C03633=1021.085,424.714,339.079,174.416,50.425,160.512
C03634=1021.073,424.470,339.128,174.401,50.423,160.509
C03635=1021.061,424.224,339.178,174.386,50.421,160.506
C03636=1021.049,423.980,339.226,174.371,50.419,160.503
C03637=1021.037,423.735,339.276,174.356,50.417,160.500
C03638=1021.025,423.490,339.323,174.341,50.416,160.496
C03639=1021.013,423.245,339.372,174.326,50.414,160.493
C03640=1021.001,422.999,339.422,174.311,50.412,160.490
C03641=1020.989,422.755,339.470,174.297,50.410,160.487
C03642=1020.978,422.510,339.519,174.282,50.409,160.484
C03643=1020.966,422.265,339.567,174.267,50.407,160.481
C03644=1020.954,422.020,339.616,174.252,50.406,160.478
C03645=1020.942,421.775,339.664,174.237,50.404,160.475
C03646=1020.931,421.530,339.713,174.223,50.402,160.472
C03647=1020.920,421.285,339.761,174.209,50.400,160.469
C03648=1020.907,421.040,339.810,174.194,50.399,160.466
C03649=1020.895,420.794,339.858,174.179,50.397,160.463
C03650=1020.884,420.549,339.906,174.165,50.396,160.460
C03651=1020.872,420.304,339.954,174.150,50.395,160.458
C03652=1020.861,420.059,340.002,174.136,50.393,160.455
C03653=1020.849,419.814,340.050,174.122,50.391,160.452
C03654=1020.837,419.569,340.098,174.108,50.390,160.449
C03655=1020.826,419.324,340.146,174.094,50.388,160.446
C03656=1020.814,419.079,340.194,174.079,50.387,160.443
C03657=1020.803,418.833,340.241,174.065,50.386,160.440
C03658=1020.791,418.588,340.289,174.051,50.384,160.437
C03659=1020.780,418.343,340.337,174.037,50.383,160.435
C03660=1020.768,418.098,340.384,174.023,50.381,160.432
C03661=1020.757,417.853,340.433,174.009,50.380,160.429
C03662=1020.746,417.607,340.480,173.995,50.378,160.426
C03663=1020.734,417.362,340.527,173.981,50.377,160.423
C03664=1020.723,417.117,340.575,173.967,50.376,160.421
C03665=1020.712,416.872,340.622,173.954,50.374,160.418
C03666=1020.701,416.626,340.671,173.940,50.373,160.415
C03667=1020.690,416.381,340.717,173.926,50.372,160.412
C03668=1020.678,416.136,340.765,173.913,50.370,160.410
C03669=1020.667,415.890,340.813,173.898,50.369,160.407
C03670=1020.656,415.645,340.859,173.885,50.368,160.404
C03671=1020.644,415.400,340.907,173.872,50.366,160.401
C03672=1020.634,415.155,340.954,173.858,50.365,160.399
C03673=1020.623,414.909,341.001,173.844,50.364,160.396
C03674=1020.612,414.664,341.048,173.831,50.363,160.394
C03675=1020.600,414.419,341.095,173.818,50.362,160.391
C03676=1020.589,414.174,341.141,173.803,50.360,160.388
C03677=1020.578,413.928,341.188,173.790,50.359,160.386
C03678=1020.568,413.683,341.235,173.777,50.358,160.383
C03679=1020.556,413.437,341.282,173.764,50.357,160.381
C03680=1020.545,413.192,341.328,173.751,50.356,160.378
C03681=1020.535,412.947,341.375,173.738,50.355,160.375
C03682=1020.519,412.599,341.441,173.719,50.353,160.372
C03683=1020.503,412.251,341.507,173.700,50.352,160.368
C03684=1020.488,411.903,341.573,173.682,50.351,160.365
C03685=1020.472,411.556,341.639,173.663,50.349,160.361
C03686=1020.461,411.311,341.685,173.651,50.348,160.359
C03687=1020.451,411.065,341.731,173.637,50.347,160.356
C03688=1020.440,410.820,341.777,173.624,50.346,160.353
C03689=1020.430,410.574,341.824,173.611,50.345,160.351
C03690=1020.419,410.329,341.870,173.599,50.344,160.349
C03691=1020.409,410.083,341.916,173.586,50.343,160.346
C03692=1020.398,409.838,341.963,173.573,50.342,160.344
C03693=1020.387,409.592,342.009,173.561,50.341,160.341
C03694=1020.376,409.347,342.055,173.548,50.340,160.339
C03695=1020.366,409.101,342.100,173.535,50.340,160.336
C03696=1020.355,408.856,342.146,173.523,50.338,160.334
C03697=1020.345,408.610,342.192,173.510,50.338,160.332
C03698=1020.334,408.365,342.238,173.497,50.337,160.329
C03699=1020.323,408.119,342.284,173.484,50.336,160.327
C03700=1020.312,407.873,342.329,173.473,50.335,160.324
C03701=1020.302,407.627,342.375,173.460,50.335,160.322
C03702=1020.291,407.382,342.421,173.447,50.334,160.320
C03703=1020.281,407.137,342.466,173.434,50.334,160.317
C03704=1020.271,406.891,342.511,173.423,50.333,160.315
C03705=1020.259,406.645,342.557,173.410,50.332,160.313
C03706=1020.249,406.399,342.602,173.398,50.331,160.311
C03707=1020.239,406.154,342.647,173.386,50.331,160.308
C03708=1020.229,405.908,342.692,173.373,50.330,160.306
C03709=1020.217,405.663,342.738,173.361,50.329,160.304
C03710=1020.208,405.417,342.783,173.349,50.329,160.301
C03711=1020.197,405.172,342.829,173.337,50.328,160.299
C03712=1020.187,404.926,342.873,173.324,50.327,160.297
C03713=1020.177,404.680,342.919,173.313,50.327,160.295
C03714=1020.166,404.435,342.963,173.300,50.326,160.292
C03715=1020.156,404.189,343.009,173.288,50.325,160.290
C03716=1020.146,403.944,343.053,173.276,50.325,160.288
C03717=1020.136,403.697,343.099,173.264,50.324,160.286
C03718=1020.125,403.452,343.143,173.253,50.324,160.284
C03719=1020.115,403.206,343.188,173.240,50.323,160.281
C03720=1020.105,402.961,343.233,173.229,50.323,160.279
C03721=1020.096,402.715,343.278,173.216,50.323,160.277
C03722=1020.085,402.469,343.323,173.205,50.322,160.275
C03723=1020.075,402.224,343.367,173.193,50.321,160.273
C03724=1020.065,401.978,343.412,173.181,50.321,160.271
C03725=1020.055,401.733,343.457,173.169,50.320,160.268
C03726=1020.045,401.486,343.502,173.158,50.320,160.266
C03727=1020.035,401.241,343.546,173.147,50.320,160.264
C03728=1020.025,400.995,343.590,173.134,50.320,160.262
C03729=1020.016,400.750,343.635,173.123,50.319,160.260
C03730=1020.006,400.503,343.679,173.111,50.318,160.258
C03731=1019.995,400.257,343.724,173.100,50.318,160.256
C03732=1019.986,400.011,343.768,173.088,50.318,160.254
C03733=1019.976,399.766,343.813,173.076,50.318,160.252
C03734=1019.966,399.520,343.856,173.065,50.317,160.250
C03735=1019.956,399.275,343.901,173.054,50.317,160.248
C03736=1019.946,399.029,343.945,173.042,50.316,160.246
C03737=1019.937,398.783,343.989,173.031,50.316,160.244
C03738=1019.927,398.537,344.034,173.020,50.316,160.242
C03739=1019.917,398.291,344.077,173.008,50.316,160.240
C03740=1019.907,398.045,344.121,172.997,50.316,160.238
C03741=1019.897,397.799,344.165,172.985,50.316,160.236
C03742=1019.885,397.475,344.223,172.971,50.316,160.233
C03743=1019.872,397.150,344.280,172.955,50.315,160.231
C03744=1019.858,396.825,344.338,172.941,50.315,160.228
C03745=1019.846,396.500,344.396,172.926,50.315,160.226
C03746=1019.836,396.254,344.440,172.915,50.315,160.224
C03747=1019.826,396.009,344.483,172.904,50.315,160.222
C03748=1019.816,395.762,344.527,172.892,50.315,160.220
C03749=1019.807,395.516,344.570,172.882,50.315,160.218
C03750=1019.798,395.271,344.614,172.871,50.314,160.216
C03751=1019.788,395.025,344.657,172.860,50.314,160.214
C03752=1019.777,394.779,344.701,172.849,50.315,160.212
C03753=1019.768,394.532,344.744,172.838,50.315,160.211
C03754=1019.759,394.287,344.787,172.827,50.314,160.208
C03755=1019.749,394.041,344.830,172.816,50.314,160.207
C03756=1019.740,393.794,344.874,172.805,50.315,160.205
C03757=1019.730,393.549,344.917,172.794,50.315,160.203
C03758=1019.721,393.303,344.961,172.783,50.315,160.201
C03759=1019.711,393.056,345.003,172.773,50.315,160.200
C03760=1019.702,392.810,345.046,172.763,50.315,160.198
C03761=1019.692,392.564,345.090,172.751,50.315,160.196
C03762=1019.683,392.318,345.132,172.740,50.315,160.194
C03763=1019.673,392.072,345.175,172.730,50.316,160.192
C03764=1019.664,391.826,345.218,172.720,50.315,160.191
C03765=1019.655,391.580,345.261,172.709,50.316,160.189
C03766=1019.645,391.334,345.304,172.698,50.316,160.187
C03767=1019.636,391.088,345.347,172.687,50.316,160.185
C03768=1019.626,390.842,345.389,172.677,50.316,160.183
C03769=1019.616,390.596,345.432,172.667,50.317,160.182
C03770=1019.608,390.350,345.475,172.656,50.317,160.180
C03771=1019.599,390.103,345.517,172.645,50.317,160.178
C03772=1019.589,389.857,345.560,172.635,50.317,160.177
C03773=1019.580,389.611,345.602,172.624,50.318,160.175
C03774=1019.571,389.365,345.645,172.614,50.317,160.173
C03775=1019.562,389.119,345.688,172.604,50.318,160.171
C03776=1019.552,388.873,345.730,172.593,50.318,160.170
C03777=1019.543,388.627,345.772,172.583,50.319,160.168
C03778=1019.534,388.380,345.815,172.572,50.319,160.166
C03779=1019.524,388.134,345.857,172.562,50.320,160.165
C03780=1019.515,387.888,345.899,172.552,50.319,160.163
C03781=1019.506,387.642,345.942,172.541,50.320,160.161
C03782=1019.497,387.395,345.984,172.532,50.321,160.160
C03783=1019.488,387.149,346.027,172.521,50.321,160.158
C03784=1019.479,386.903,346.068,172.511,50.321,160.156
C03785=1019.470,386.656,346.110,172.501,50.322,160.155
C03786=1019.461,386.411,346.153,172.490,50.323,160.153
C03787=1019.452,386.164,346.194,172.481,50.323,160.152
C03788=1019.443,385.918,346.236,172.470,50.323,160.150
C03789=1019.434,385.672,346.278,172.460,50.324,160.148
C03790=1019.425,385.426,346.320,172.451,50.324,160.147
C03791=1019.416,385.179,346.362,172.440,50.325,160.145
C03792=1019.407,384.932,346.404,172.431,50.325,160.144
C03793=1019.397,384.686,346.445,172.420,50.326,160.142
C03794=1019.388,384.440,346.487,172.410,50.326,160.141
C03795=1019.379,384.194,346.528,172.400,50.327,160.139
C03796=1019.370,383.947,346.570,172.391,50.328,160.138
C03797=1019.361,383.701,346.612,172.380,50.329,160.136
C03798=1019.351,383.455,346.653,172.371,50.329,160.135
C03799=1019.343,383.209,346.694,172.360,50.330,160.133
C03800=1019.335,382.962,346.735,172.351,50.330,160.132
C03801=1019.326,382.716,346.777,172.341,50.331,160.130
C03802=1019.314,382.429,346.826,172.329,50.332,160.128
C03803=1019.304,382.141,346.873,172.318,50.333,160.127
C03804=1019.294,381.854,346.921,172.306,50.334,160.125
C03805=1019.283,381.567,346.970,172.296,50.335,160.123
C03806=1019.275,381.321,347.011,172.285,50.336,160.122
C03807=1019.266,381.074,347.052,172.276,50.336,160.120
C03808=1019.257,380.828,347.094,172.267,50.337,160.119
C03809=1019.248,380.581,347.135,172.256,50.338,160.117
C03810=1019.239,380.335,347.176,172.247,50.339,160.116
C03811=1019.231,380.088,347.217,172.238,50.340,160.115
C03812=1019.222,379.841,347.258,172.228,50.340,160.113
C03813=1019.214,379.596,347.299,172.218,50.341,160.112
C03814=1019.205,379.349,347.340,172.208,50.342,160.110
C03815=1019.196,379.102,347.380,172.199,50.343,160.109
C03816=1019.188,378.857,347.422,172.190,50.344,160.108
C03817=1019.179,378.610,347.463,172.180,50.344,160.106
C03818=1019.171,378.363,347.503,172.170,50.345,160.105
C03819=1019.162,378.117,347.545,172.161,50.346,160.103
C03820=1019.153,377.871,347.585,172.152,50.347,160.102
C03821=1019.145,377.624,347.626,172.143,50.348,160.101
C03822=1019.137,377.378,347.667,172.133,50.349,160.099
C03823=1019.128,377.131,347.708,172.123,50.350,160.098
C03824=1019.119,376.885,347.748,172.114,50.351,160.097
C03825=1019.110,376.638,347.789,172.105,50.352,160.095
C03826=1019.102,376.391,347.830,172.096,50.353,160.094
C03827=1019.094,376.144,347.871,172.087,50.354,160.093
C03828=1019.086,375.898,347.911,172.077,50.355,160.091
C03829=1019.076,375.651,347.952,172.068,50.356,160.090
C03830=1019.068,375.405,347.992,172.059,50.357,160.089
C03831=1019.060,375.159,348.032,172.050,50.358,160.087
C03832=1019.051,374.912,348.072,172.040,50.359,160.086
C03833=1019.043,374.666,348.113,172.031,50.361,160.085
C03834=1019.034,374.418,348.152,172.022,50.362,160.084
C03835=1019.025,374.172,348.193,172.013,50.363,160.082
C03836=1019.017,373.925,348.232,172.003,50.364,160.081
C03837=1019.009,373.679,348.273,171.995,50.365,160.080
C03838=1019.000,373.432,348.313,171.986,50.366,160.079
C03839=1018.991,373.186,348.353,171.976,50.367,160.077
C03840=1018.983,372.939,348.392,171.968,50.369,160.076
C03841=1018.974,372.692,348.433,171.958,50.370,160.075
C03842=1018.966,372.445,348.473,171.950,50.372,160.074
C03843=1018.958,372.199,348.513,171.940,50.372,160.072
C03844=1018.950,371.953,348.553,171.932,50.374,160.071
C03845=1018.941,371.706,348.592,171.923,50.375,160.070
C03846=1018.933,371.460,348.633,171.914,50.377,160.069
C03847=1018.924,371.212,348.672,171.905,50.378,160.068
C03848=1018.916,370.966,348.712,171.896,50.379,160.067
C03849=1018.908,370.719,348.752,171.887,50.380,160.065
C03850=1018.899,370.473,348.792,171.878,50.382,160.064
C03851=1018.892,370.226,348.832,171.869,50.383,160.063
C03852=1018.883,369.979,348.871,171.860,50.384,160.062
C03853=1018.876,369.732,348.911,171.851,50.386,160.061
C03854=1018.867,369.486,348.950,171.842,50.387,160.059
C03855=1018.859,369.239,348.990,171.834,50.388,160.058
C03856=1018.851,368.992,349.029,171.825,50.390,160.057
C03857=1018.842,368.746,349.069,171.817,50.391,160.056
C03858=1018.835,368.499,349.109,171.808,50.393,160.055
C03859=1018.826,368.252,349.148,171.799,50.394,160.054
C03860=1018.819,368.005,349.188,171.790,50.395,160.053
C03861=1018.810,367.759,349.227,171.781,50.397,160.051
C03862=1018.801,367.494,349.269,171.772,50.398,160.050
C03863=1018.793,367.229,349.311,171.763,50.400,160.049
C03864=1018.784,366.963,349.353,171.754,50.402,160.048
C03865=1018.775,366.699,349.396,171.745,50.404,160.047
C03866=1018.767,366.452,349.434,171.736,50.405,160.046
C03867=1018.759,366.205,349.473,171.727,50.407,160.045
C03868=1018.750,365.958,349.512,171.719,50.408,160.044
C03869=1018.743,365.712,349.551,171.710,50.410,160.043
C03870=1018.734,365.465,349.590,171.701,50.411,160.041
C03871=1018.727,365.218,349.630,171.693,50.413,160.040
C03872=1018.719,364.971,349.668,171.685,50.415,160.040
C03873=1018.710,364.724,349.707,171.676,50.416,160.038
C03874=1018.703,364.477,349.746,171.667,50.418,160.037
C03875=1018.694,364.230,349.784,171.659,50.420,160.036
C03876=1018.686,363.984,349.824,171.651,50.421,160.035
C03877=1018.678,363.737,349.862,171.642,50.423,160.034
C03878=1018.670,363.490,349.900,171.634,50.425,160.033
C03879=1018.662,363.243,349.940,171.625,50.427,160.032
C03880=1018.654,362.997,349.978,171.617,50.428,160.031
C03881=1018.647,362.749,350.017,171.609,50.430,160.030
C03882=1018.639,362.502,350.056,171.600,50.432,160.029
C03883=1018.631,362.256,350.094,171.591,50.433,160.028
C03884=1018.623,362.009,350.133,171.584,50.435,160.027
C03885=1018.615,361.762,350.172,171.575,50.437,160.026
C03886=1018.607,361.515,350.210,171.567,50.439,160.025
C03887=1018.599,361.268,350.249,171.560,50.441,160.025
C03888=1018.591,361.022,350.287,171.551,50.442,160.023
C03889=1018.583,360.774,350.326,171.542,50.445,160.023
C03890=1018.577,360.563,350.359,171.536,50.445,160.022
C03891=1018.571,360.352,350.391,171.528,50.447,160.021
C03892=1018.564,360.142,350.425,171.522,50.449,160.020
C03893=1018.557,359.931,350.457,171.514,50.451,160.019
C03894=1018.550,359.720,350.490,171.508,50.452,160.019
C03895=1018.544,359.509,350.522,171.501,50.454,160.018
C03896=1018.538,359.299,350.555,171.494,50.455,160.017
C03897=1018.531,359.088,350.587,171.487,50.457,160.016
C03898=1018.523,358.841,350.625,171.478,50.459,160.015
C03899=1018.515,358.595,350.664,171.471,50.461,160.014
C03900=1018.507,358.347,350.702,171.462,50.463,160.013
C03901=1018.500,358.100,350.740,171.455,50.465,160.013
C03902=1018.492,357.853,350.778,171.446,50.467,160.012
C03903=1018.484,357.606,350.816,171.438,50.469,160.011
C03904=1018.476,357.360,350.854,171.431,50.471,160.010
C03905=1018.468,357.112,350.892,171.422,50.473,160.009
C03906=1018.461,356.865,350.930,171.414,50.475,160.008
C03907=1018.453,356.618,350.967,171.406,50.477,160.007
C03908=1018.445,356.371,351.006,171.398,50.479,160.006
C03909=1018.437,356.124,351.043,171.391,50.481,160.006
C03910=1018.430,355.877,351.080,171.382,50.483,160.005
C03911=1018.423,355.631,351.119,171.374,50.485,160.004
C03912=1018.415,355.383,351.157,171.366,50.487,160.003
C03913=1018.407,355.136,351.193,171.358,50.490,160.002
C03914=1018.399,354.889,351.232,171.351,50.492,160.001
C03915=1018.392,354.642,351.269,171.343,50.494,160.001
C03916=1018.385,354.395,351.307,171.335,50.496,160.000
C03917=1018.376,354.148,351.344,171.327,50.498,159.999
C03918=1018.369,353.900,351.382,171.320,50.501,159.998
C03919=1018.361,353.654,351.420,171.311,50.503,159.997
C03920=1018.354,353.407,351.457,171.304,50.505,159.997
C03921=1018.346,353.160,351.494,171.296,50.508,159.996
C03922=1018.336,352.830,351.543,171.286,50.510,159.995
C03923=1018.326,352.500,351.594,171.275,50.513,159.994
C03924=1018.315,352.170,351.644,171.265,50.516,159.993
C03925=1018.305,351.840,351.694,171.255,50.520,159.992
C03926=1018.298,351.592,351.730,171.246,50.522,159.991
C03927=1018.290,351.346,351.767,171.239,50.524,159.990
C03928=1018.283,351.098,351.805,171.231,50.527,159.989
C03929=1018.276,350.851,351.842,171.224,50.529,159.989
C03930=1018.268,350.604,351.879,171.216,50.531,159.988
C03931=1018.261,350.357,351.916,171.209,50.534,159.987
C03932=1018.253,350.110,351.953,171.200,50.536,159.986
C03933=1018.246,349.863,351.991,171.193,50.538,159.986
C03934=1018.238,349.616,352.027,171.185,50.541,159.985
C03935=1018.231,349.368,352.064,171.178,50.543,159.984
C03936=1018.223,349.121,352.102,171.171,50.545,159.984
C03937=1018.216,348.874,352.138,171.163,50.548,159.983
C03938=1018.209,348.627,352.175,171.156,50.551,159.982
C03939=1018.201,348.380,352.212,171.147,50.553,159.981
C03940=1018.194,348.133,352.249,171.140,50.555,159.981
C03941=1018.186,347.886,352.286,171.132,50.558,159.980
C03942=1018.179,347.638,352.323,171.125,50.561,159.980
C03943=1018.171,347.391,352.360,171.118,50.563,159.979
C03944=1018.165,347.144,352.396,171.110,50.565,159.978
C03945=1018.157,346.897,352.433,171.103,50.568,159.977
C03946=1018.150,346.650,352.470,171.095,50.571,159.977
C03947=1018.142,346.402,352.506,171.088,50.573,159.976
C03948=1018.135,346.155,352.542,171.080,50.576,159.975
C03949=1018.128,345.908,352.579,171.073,50.578,159.975
C03950=1018.120,345.661,352.616,171.066,50.581,159.974
C03951=1018.113,345.413,352.652,171.058,50.584,159.973
C03952=1018.106,345.166,352.688,171.051,50.586,159.973
C03953=1018.099,344.919,352.725,171.043,50.589,159.972
C03954=1018.091,344.672,352.761,171.036,50.592,159.972
C03955=1018.083,344.425,352.798,171.029,50.594,159.971
C03956=1018.077,344.178,352.834,171.021,50.597,159.970
C03957=1018.069,343.930,352.870,171.014,50.600,159.970
C03958=1018.061,343.683,352.907,171.006,50.603,159.969
C03959=1018.055,343.436,352.943,170.999,50.605,159.969
C03960=1018.047,343.188,352.979,170.992,50.608,159.968
C03961=1018.040,342.941,353.015,170.984,50.611,159.967
C03962=1018.033,342.694,353.052,170.977,50.613,159.967
C03963=1018.026,342.446,353.088,170.970,50.616,159.966
C03964=1018.018,342.199,353.124,170.963,50.619,159.966
C03965=1018.011,341.951,353.159,170.956,50.622,159.965
C03966=1018.005,341.704,353.196,170.949,50.624,159.964
C03967=1017.997,341.457,353.232,170.941,50.628,159.964
C03968=1017.990,341.210,353.268,170.934,50.630,159.963
C03969=1017.982,340.963,353.304,170.927,50.633,159.963
C03970=1017.976,340.715,353.339,170.920,50.636,159.962
C03971=1017.969,340.468,353.376,170.913,50.639,159.962
C03972=1017.962,340.221,353.412,170.906,50.642,159.961
C03973=1017.954,339.973,353.448,170.898,50.645,159.961
C03974=1017.947,339.726,353.483,170.891,50.648,159.960
C03975=1017.939,339.479,353.520,170.884,50.650,159.960
C03976=1017.933,339.231,353.555,170.877,50.654,159.959
C03977=1017.926,338.984,353.591,170.870,50.656,159.958
C03978=1017.919,338.737,353.627,170.863,50.659,159.958
C03979=1017.912,338.489,353.662,170.855,50.663,159.958
C03980=1017.905,338.241,353.698,170.848,50.665,159.957
C03981=1017.897,337.995,353.734,170.842,50.668,159.956
C03982=1017.890,337.735,353.771,170.834,50.672,159.956
C03983=1017.883,337.474,353.808,170.826,50.674,159.955
C03984=1017.875,337.214,353.845,170.819,50.678,159.955
C03985=1017.867,336.953,353.883,170.812,50.681,159.954
C03986=1017.860,336.706,353.918,170.805,50.684,159.954
C03987=1017.853,336.459,353.953,170.798,50.688,159.953
C03988=1017.846,336.211,353.989,170.791,50.690,159.953
C03989=1017.839,335.964,354.025,170.784,50.693,159.952
C03990=1017.832,335.717,354.060,170.776,50.697,159.952
C03991=1017.825,335.469,354.095,170.770,50.700,159.952
C03992=1017.818,335.221,354.131,170.763,50.703,159.951
C03993=1017.811,334.974,354.166,170.756,50.706,159.951
C03994=1017.804,334.727,354.202,170.749,50.709,159.950
C03995=1017.797,334.480,354.237,170.742,50.713,159.950
C03996=1017.790,334.232,354.272,170.736,50.716,159.949
C03997=1017.783,333.984,354.307,170.729,50.719,159.949
C03998=1017.777,333.737,354.342,170.721,50.722,159.949
C03999=1017.770,333.490,354.378,170.715,50.725,159.948
C04000=1017.763,333.242,354.413,170.708,50.728,159.948
C04001=1017.756,332.995,354.448,170.702,50.732,159.947
C04002=1017.749,332.747,354.483,170.694,50.735,159.947
C04003=1017.741,332.500,354.518,170.687,50.738,159.946
C04004=1017.735,332.252,354.553,170.681,50.741,159.946
C04005=1017.728,332.005,354.588,170.674,50.744,159.946
C04006=1017.721,331.757,354.623,170.666,50.748,159.945
C04007=1017.714,331.510,354.657,170.660,50.752,159.945
C04008=1017.707,331.263,354.692,170.654,50.755,159.944
C04009=1017.700,331.015,354.727,170.647,50.758,159.944
C04010=1017.693,330.768,354.761,170.639,50.761,159.944
C04011=1017.686,330.520,354.796,170.633,50.765,159.943
C04012=1017.680,330.273,354.831,170.626,50.768,159.943
C04013=1017.672,330.025,354.865,170.620,50.771,159.943
C04014=1017.666,329.778,354.900,170.613,50.775,159.942
C04015=1017.659,329.530,354.936,170.606,50.779,159.942
C04016=1017.652,329.282,354.970,170.599,50.782,159.941
C04017=1017.645,329.035,355.005,170.593,50.785,159.941
C04018=1017.638,328.787,355.039,170.586,50.789,159.941
C04019=1017.632,328.540,355.074,170.579,50.792,159.940
C04020=1017.624,328.292,355.108,170.573,50.796,159.940
C04021=1017.618,328.045,355.143,170.566,50.799,159.940
C04022=1017.611,327.797,355.177,170.560,50.803,159.939
C04023=1017.604,327.550,355.212,170.552,50.806,159.939
C04024=1017.598,327.303,355.246,170.546,50.810,159.939
C04025=1017.591,327.055,355.281,170.539,50.813,159.938
C04026=1017.584,326.808,355.315,170.533,50.817,159.938
C04027=1017.577,326.560,355.349,170.526,50.820,159.938
C04028=1017.571,326.312,355.385,170.519,50.824,159.937
C04029=1017.563,326.065,355.418,170.513,50.828,159.937
C04030=1017.557,325.818,355.452,170.506,50.831,159.937
C04031=1017.550,325.570,355.486,170.500,50.835,159.937
C04032=1017.543,325.322,355.520,170.493,50.839,159.936
C04033=1017.536,325.075,355.555,170.487,50.843,159.936
C04034=1017.529,324.827,355.588,170.480,50.846,159.936
C04035=1017.522,324.579,355.623,170.474,50.849,159.935
C04036=1017.515,324.332,355.656,170.467,50.854,159.935
C04037=1017.508,324.085,355.690,170.460,50.857,159.935
C04038=1017.501,323.837,355.724,170.454,50.861,159.935
C04039=1017.495,323.589,355.758,170.448,50.865,159.935
C04040=1017.488,323.342,355.792,170.441,50.869,159.934
C04041=1017.481,323.094,355.825,170.434,50.872,159.934
C04042=1017.474,322.829,355.862,170.427,50.877,159.934
C04043=1017.466,322.565,355.898,170.421,50.881,159.934
C04044=1017.459,322.300,355.934,170.414,50.885,159.933
C04045=1017.452,322.035,355.970,170.407,50.889,159.933
C04046=1017.445,321.788,356.004,170.400,50.893,159.933
C04047=1017.438,321.540,356.037,170.394,50.896,159.933
C04048=1017.431,321.292,356.071,170.388,50.900,159.932
C04049=1017.425,321.045,356.105,170.381,50.904,159.932
C04050=1017.418,320.798,356.139,170.375,50.908,159.932
C04051=1017.412,320.550,356.171,170.368,50.912,159.932
C04052=1017.405,320.302,356.205,170.362,50.916,159.931
C04053=1017.397,320.055,356.239,170.356,50.919,159.931
C04054=1017.392,319.807,356.273,170.349,50.924,159.931
C04055=1017.385,319.559,356.306,170.342,50.927,159.931
C04056=1017.378,319.312,356.340,170.337,50.932,159.931
C04057=1017.371,319.064,356.373,170.330,50.936,159.930
C04058=1017.365,318.816,356.407,170.324,50.939,159.930
C04059=1017.358,318.569,356.441,170.317,50.943,159.930
C04060=1017.352,318.321,356.473,170.311,50.947,159.930
C04061=1017.345,318.074,356.507,170.305,50.952,159.930
C04062=1017.339,317.826,356.541,170.299,50.955,159.930
C04063=1017.332,317.578,356.574,170.292,50.959,159.929
C04064=1017.325,317.331,356.608,170.286,50.963,159.929
C04065=1017.318,317.083,356.641,170.279,50.968,159.929
C04066=1017.312,316.836,356.674,170.273,50.972,159.929
C04067=1017.306,316.588,356.708,170.267,50.975,159.929
C04068=1017.299,316.340,356.741,170.261,50.980,159.929
C04069=1017.293,316.093,356.774,170.255,50.984,159.928
C04070=1017.286,315.844,356.807,170.249,50.987,159.928
C04071=1017.280,315.597,356.841,170.242,50.992,159.928
C04072=1017.274,315.349,356.874,170.236,50.996,159.928
C04073=1017.267,315.101,356.907,170.230,51.000,159.928
C04074=1017.260,314.854,356.941,170.224,51.004,159.928
C04075=1017.254,314.607,356.974,170.217,51.008,159.927
C04076=1017.248,314.359,357.007,170.212,51.012,159.927
C04077=1017.241,314.111,357.041,170.205,51.016,159.927
C04078=1017.235,313.863,357.073,170.198,51.021,159.927
C04079=1017.229,313.616,357.106,170.192,51.025,159.927
C04080=1017.221,313.368,357.140,170.186,51.029,159.927
C04081=1017.216,313.120,357.173,170.180,51.033,159.927
C04082=1017.209,312.873,357.206,170.174,51.037,159.927
C04083=1017.203,312.625,357.239,170.169,51.042,159.927
C04084=1017.197,312.377,357.272,170.162,51.046,159.926
C04085=1017.190,312.130,357.305,170.157,51.050,159.926
C04086=1017.184,311.882,357.339,170.150,51.054,159.926
C04087=1017.178,311.634,357.371,170.143,51.059,159.926
C04088=1017.172,311.387,357.404,170.138,51.063,159.926
C04089=1017.165,311.139,357.437,170.131,51.067,159.926
C04090=1017.159,310.891,357.470,170.126,51.071,159.926
C04091=1017.153,310.644,357.503,170.120,51.076,159.926
C04092=1017.147,310.395,357.536,170.114,51.080,159.926
C04093=1017.140,310.148,357.569,170.108,51.084,159.926
C04094=1017.134,309.900,357.602,170.102,51.089,159.926
C04095=1017.128,309.652,357.634,170.096,51.092,159.925
C04096=1017.121,309.405,357.667,170.089,51.097,159.925
C04097=1017.115,309.157,357.700,170.083,51.102,159.925
C04098=1017.108,308.909,357.731,170.077,51.106,159.925
C04099=1017.102,308.662,357.764,170.071,51.110,159.925
C04100=1017.095,308.415,357.796,170.066,51.115,159.925
C04101=1017.089,308.166,357.828,170.059,51.120,159.925
C04102=1017.082,307.907,357.862,170.053,51.125,159.925
C04103=1017.075,307.648,357.896,170.047,51.130,159.925
C04104=1017.068,307.389,357.929,170.041,51.134,159.925
C04105=1017.061,307.130,357.963,170.034,51.139,159.925
C04106=1017.055,306.882,357.995,170.028,51.143,159.925
C04107=1017.048,306.634,358.028,170.022,51.148,159.925
C04108=1017.042,306.386,358.060,170.017,51.153,159.925
C04109=1017.035,306.139,358.092,170.010,51.158,159.925
C04110=1017.029,305.891,358.124,170.004,51.162,159.925
C04111=1017.022,305.643,358.156,169.998,51.167,159.925
C04112=1017.016,305.395,358.188,169.993,51.171,159.925
C04113=1017.010,305.147,358.220,169.987,51.176,159.925
C04114=1017.003,304.900,358.252,169.980,51.181,159.925
C04115=1016.997,304.651,358.284,169.975,51.186,159.925
C04116=1016.990,304.404,358.316,169.969,51.190,159.925
C04117=1016.984,304.156,358.348,169.963,51.195,159.925
C04118=1016.977,303.908,358.380,169.958,51.200,159.925
C04119=1016.971,303.660,358.412,169.951,51.204,159.925
C04120=1016.965,303.412,358.445,169.945,51.209,159.925
C04121=1016.959,303.165,358.476,169.940,51.214,159.925
C04122=1016.953,302.917,358.508,169.934,51.218,159.925
C04123=1016.946,302.670,358.540,169.928,51.223,159.925
C04124=1016.940,302.421,358.572,169.921,51.228,159.926
C04125=1016.933,302.173,358.603,169.916,51.233,159.926
C04126=1016.927,301.925,358.635,169.910,51.238,159.926
C04127=1016.920,301.677,358.667,169.904,51.243,159.926
C04128=1016.915,301.430,358.698,169.899,51.247,159.926
C04129=1016.908,301.183,358.731,169.893,51.252,159.926
C04130=1016.902,300.934,358.763,169.886,51.257,159.926
C04131=1016.896,300.686,358.795,169.881,51.262,159.926
C04132=1016.889,300.438,358.826,169.875,51.267,159.926
C04133=1016.884,300.191,358.858,169.870,51.272,159.926
C04134=1016.877,299.943,358.889,169.864,51.276,159.926
C04135=1016.871,299.695,358.921,169.859,51.281,159.926
C04136=1016.865,299.447,358.953,169.852,51.286,159.926
C04137=1016.859,299.199,358.984,169.846,51.291,159.926
C04138=1016.852,298.951,359.016,169.841,51.296,159.927
C04139=1016.846,298.703,359.048,169.835,51.301,159.927
C04140=1016.840,298.455,359.079,169.830,51.306,159.927
C04141=1016.834,298.208,359.111,169.824,51.311,159.927
C04142=1016.828,297.959,359.143,169.818,51.316,159.927
C04143=1016.822,297.712,359.174,169.812,51.321,159.927
C04144=1016.816,297.464,359.206,169.806,51.326,159.927
C04145=1016.809,297.216,359.237,169.801,51.331,159.927
C04146=1016.803,296.968,359.269,169.796,51.336,159.927
C04147=1016.798,296.720,359.300,169.790,51.340,159.927
C04148=1016.792,296.472,359.332,169.783,51.346,159.927
C04149=1016.786,296.225,359.363,169.778,51.351,159.928
C04150=1016.780,295.976,359.395,169.772,51.356,159.928
C04151=1016.773,295.729,359.426,169.767,51.361,159.928
C04152=1016.767,295.481,359.458,169.761,51.366,159.928
C04153=1016.761,295.233,359.489,169.756,51.371,159.928
C04154=1016.756,294.985,359.520,169.751,51.376,159.928
C04155=1016.750,294.737,359.552,169.744,51.381,159.928
C04156=1016.744,294.490,359.583,169.738,51.386,159.928
C04157=1016.738,294.241,359.615,169.733,51.391,159.929
C04158=1016.732,293.997,359.646,169.728,51.396,159.929
C04159=1016.726,293.752,359.676,169.722,51.402,159.929
C04160=1016.720,293.507,359.707,169.716,51.406,159.929
C04161=1016.714,293.262,359.739,169.711,51.411,159.929
C04162=1016.708,293.018,359.769,169.706,51.416,159.929
C04163=1016.702,292.773,359.800,169.700,51.422,159.930
C04164=1016.696,292.529,359.830,169.695,51.427,159.930
C04165=1016.690,292.284,359.861,169.689,51.432,159.930
C04166=1016.684,292.037,359.892,169.683,51.437,159.930
C04167=1016.678,291.789,359.922,169.678,51.443,159.930
C04168=1016.672,291.540,359.954,169.672,51.448,159.930
C04169=1016.666,291.293,359.985,169.667,51.453,159.931
C04170=1016.660,291.044,360.016,169.662,51.459,159.931
C04171=1016.654,290.796,360.046,169.655,51.464,159.931
C04172=1016.647,290.548,360.077,169.650,51.469,159.931
C04173=1016.641,290.301,360.108,169.645,51.475,159.932
C04174=1016.636,290.053,360.138,169.639,51.480,159.932
C04175=1016.629,289.804,360.169,169.633,51.486,159.932
C04176=1016.623,289.557,360.200,169.628,51.491,159.932
C04177=1016.617,289.309,360.231,169.622,51.496,159.932
C04178=1016.612,289.060,360.262,169.617,51.501,159.933
C04179=1016.606,288.813,360.292,169.611,51.508,159.933
C04180=1016.599,288.564,360.323,169.606,51.513,159.933
C04181=1016.593,288.316,360.353,169.600,51.518,159.933
C04182=1016.587,288.068,360.384,169.595,51.524,159.934
C04183=1016.581,287.821,360.415,169.589,51.529,159.934
C04184=1016.575,287.573,360.445,169.584,51.534,159.934
C04185=1016.569,287.324,360.476,169.579,51.540,159.934
C04186=1016.563,287.076,360.506,169.573,51.545,159.934
C04187=1016.557,286.829,360.536,169.567,51.552,159.935
C04188=1016.551,286.580,360.567,169.562,51.557,159.935
C04189=1016.545,286.332,360.598,169.557,51.563,159.935
C04190=1016.539,286.084,360.628,169.552,51.568,159.936
C04191=1016.533,285.837,360.658,169.546,51.574,159.936
C04192=1016.527,285.588,360.689,169.540,51.579,159.936
C04193=1016.521,285.340,360.719,169.535,51.585,159.936
C04194=1016.515,285.092,360.749,169.530,51.590,159.937
C04195=1016.509,284.843,360.780,169.524,51.596,159.937
C04196=1016.503,284.595,360.810,169.518,51.602,159.937
C04197=1016.497,284.348,360.840,169.513,51.608,159.938
C04198=1016.491,284.100,360.870,169.508,51.613,159.938
C04199=1016.485,283.852,360.900,169.502,51.619,159.938
C04200=1016.479,283.603,360.930,169.497,51.625,159.938
C04201=1016.472,283.356,360.960,169.492,51.631,159.939
C04202=1016.467,283.107,360.990,169.486,51.636,159.939
C04203=1016.461,282.859,361.020,169.481,51.642,159.939
C04204=1016.455,282.611,361.051,169.476,51.648,159.940
C04205=1016.448,282.363,361.080,169.470,51.653,159.940
C04206=1016.443,282.115,361.110,169.465,51.659,159.940
C04207=1016.437,281.867,361.141,169.460,51.665,159.941
C04208=1016.431,281.619,361.170,169.455,51.671,159.941
C04209=1016.425,281.371,361.200,169.449,51.677,159.941
C04210=1016.419,281.122,361.230,169.443,51.682,159.941
C04211=1016.413,280.874,361.260,169.438,51.688,159.942
C04212=1016.406,280.626,361.289,169.432,51.695,159.942
C04213=1016.401,280.378,361.320,169.427,51.700,159.942
C04214=1016.395,280.130,361.349,169.422,51.706,159.943
C04215=1016.389,279.882,361.380,169.417,51.713,159.943
C04216=1016.383,279.634,361.409,169.412,51.718,159.944
C04217=1016.377,279.386,361.439,169.407,51.724,159.944
C04218=1016.371,279.168,361.465,169.401,51.729,159.944
C04219=1016.367,278.951,361.492,169.397,51.734,159.944
C04220=1016.362,278.734,361.518,169.393,51.740,159.945
C04221=1016.356,278.517,361.544,169.388,51.745,159.945
C04222=1016.351,278.300,361.569,169.383,51.750,159.945
C04223=1016.347,278.083,361.596,169.378,51.756,159.946
C04224=1016.341,277.866,361.622,169.374,51.761,159.946
C04225=1016.332,277.478,361.668,169.366,51.770,159.947
C04226=1016.326,277.230,361.698,169.360,51.776,159.947
C04227=1016.321,276.982,361.728,169.355,51.782,159.947
C04228=1016.315,276.733,361.757,169.350,51.788,159.948
C04229=1016.309,276.486,361.787,169.344,51.794,159.948
C04230=1016.303,276.237,361.817,169.339,51.800,159.948
C04231=1016.298,275.989,361.846,169.334,51.806,159.949
C04232=1016.291,275.741,361.875,169.328,51.812,159.949
C04233=1016.285,275.493,361.905,169.324,51.819,159.950
C04234=1016.279,275.245,361.935,169.319,51.825,159.950
C04235=1016.273,274.996,361.964,169.313,51.831,159.950
C04236=1016.268,274.748,361.993,169.308,51.837,159.951
C04237=1016.261,274.500,362.022,169.303,51.844,159.951
C04238=1016.256,274.251,362.052,169.298,51.850,159.952
C04239=1016.250,274.003,362.081,169.293,51.855,159.952
C04240=1016.244,273.755,362.111,169.287,51.862,159.953
C04241=1016.238,273.507,362.139,169.282,51.868,159.953
C04242=1016.233,273.259,362.169,169.277,51.874,159.953
C04243=1016.227,273.011,362.198,169.272,51.881,159.954
C04244=1016.221,272.762,362.228,169.267,51.887,159.954
C04245=1016.215,272.514,362.257,169.261,51.893,159.955
C04246=1016.209,272.266,362.286,169.256,51.900,159.955
C04247=1016.203,272.018,362.315,169.251,51.906,159.956
C04248=1016.197,271.770,362.345,169.246,51.912,159.956
C04249=1016.192,271.522,362.374,169.241,51.919,159.956
C04250=1016.186,271.274,362.403,169.235,51.925,159.957
C04251=1016.180,271.025,362.432,169.231,51.931,159.957
C04252=1016.174,270.777,362.461,169.226,51.937,159.958
C04253=1016.168,270.528,362.490,169.220,51.944,159.958
C04254=1016.162,270.280,362.519,169.215,51.950,159.959
C04255=1016.157,270.033,362.548,169.210,51.957,159.959
C04256=1016.151,269.784,362.577,169.205,51.963,159.960
C04257=1016.145,269.535,362.606,169.199,51.970,159.960
C04258=1016.139,269.287,362.635,169.195,51.977,159.961
C04259=1016.134,269.039,362.664,169.190,51.982,159.961
C04260=1016.128,268.791,362.693,169.184,51.989,159.962
C04261=1016.122,268.543,362.722,169.179,51.995,159.962
C04262=1016.116,268.294,362.751,169.174,52.002,159.962
C04263=1016.111,268.047,362.780,169.169,52.009,159.963
C04264=1016.105,267.798,362.808,169.164,52.016,159.964
C04265=1016.099,267.550,362.837,169.159,52.022,159.964
C04266=1016.093,267.301,362.866,169.153,52.029,159.964
C04267=1016.087,267.054,362.894,169.149,52.035,159.965
C04268=1016.082,266.805,362.923,169.144,52.041,159.965
C04269=1016.076,266.556,362.952,169.138,52.048,159.966
C04270=1016.070,266.308,362.980,169.134,52.055,159.967
C04271=1016.064,266.060,363.009,169.128,52.062,159.967
C04272=1016.058,265.812,363.038,169.124,52.068,159.968
C04273=1016.053,265.564,363.067,169.118,52.075,159.968
C04274=1016.047,265.315,363.095,169.114,52.081,159.969
C04275=1016.041,265.067,363.124,169.108,52.088,159.969
C04276=1016.036,264.819,363.152,169.104,52.095,159.970
C04277=1016.029,264.571,363.181,169.098,52.102,159.970
C04278=1016.025,264.334,363.208,169.094,52.108,159.971
C04279=1016.018,264.098,363.235,169.089,52.114,159.971
C04280=1016.013,263.862,363.262,169.084,52.121,159.972
C04281=1016.008,263.625,363.290,169.080,52.127,159.972
C04282=1016.002,263.389,363.317,169.074,52.134,159.973
C04283=1015.997,263.153,363.344,169.069,52.140,159.973
C04284=1015.991,262.916,363.371,169.065,52.147,159.974
C04285=1015.986,262.680,363.398,169.060,52.154,159.974
C04286=1015.980,262.432,363.426,169.055,52.161,159.975
C04287=1015.974,262.184,363.455,169.050,52.167,159.976
C04288=1015.968,261.935,363.483,169.045,52.174,159.976
C04289=1015.963,261.687,363.511,169.040,52.181,159.977
C04290=1015.957,261.439,363.539,169.035,52.188,159.977
C04291=1015.951,261.191,363.567,169.030,52.194,159.978
C04292=1015.945,260.942,363.596,169.025,52.201,159.978
C04293=1015.941,260.694,363.625,169.020,52.208,159.979
C04294=1015.935,260.445,363.653,169.015,52.215,159.979
C04295=1015.929,260.197,363.681,169.010,52.223,159.980
C04296=1015.923,259.949,363.709,169.005,52.229,159.981
C04297=1015.918,259.701,363.737,169.000,52.236,159.981
C04298=1015.911,259.452,363.765,168.995,52.243,159.982
C04299=1015.906,259.204,363.793,168.990,52.251,159.982
C04300=1015.900,258.955,363.821,168.985,52.258,159.983
C04301=1015.894,258.708,363.849,168.980,52.264,159.984
C04302=1015.888,258.459,363.877,168.975,52.272,159.984
C04303=1015.882,258.211,363.904,168.970,52.279,159.985
C04304=1015.876,257.962,363.933,168.966,52.286,159.986
C04305=1015.871,257.714,363.960,168.960,52.293,159.986
C04306=1015.864,257.465,363.988,168.955,52.301,159.987
C04307=1015.859,257.217,364.016,168.951,52.308,159.987
C04308=1015.853,256.969,364.043,168.946,52.315,159.988
C04309=1015.847,256.720,364.071,168.940,52.322,159.989
C04310=1015.842,256.472,364.098,168.936,52.330,159.989
C04311=1015.835,256.224,364.126,168.931,52.337,159.990
C04312=1015.830,255.975,364.154,168.926,52.344,159.991
C04313=1015.824,255.726,364.182,168.921,52.351,159.991
C04314=1015.818,255.478,364.209,168.916,52.359,159.992
C04315=1015.813,255.230,364.237,168.911,52.366,159.992
C04316=1015.806,254.981,364.264,168.906,52.373,159.993
C04317=1015.801,254.733,364.292,168.902,52.381,159.994
C04318=1015.795,254.484,364.320,168.896,52.388,159.995
C04319=1015.789,254.236,364.347,168.891,52.395,159.995
C04320=1015.784,253.988,364.375,168.887,52.403,159.996
C04321=1015.777,253.740,364.403,168.882,52.410,159.997
C04322=1015.772,253.491,364.430,168.877,52.417,159.997
C04323=1015.767,253.243,364.458,168.873,52.425,159.998
C04324=1015.761,252.994,364.485,168.867,52.432,159.999
C04325=1015.755,252.746,364.513,168.862,52.440,159.999
C04326=1015.750,252.498,364.541,168.857,52.447,160.000
C04327=1015.743,252.249,364.568,168.853,52.454,160.001
C04328=1015.738,252.001,364.596,168.848,52.462,160.001
C04329=1015.732,251.752,364.623,168.843,52.469,160.002
C04330=1015.727,251.504,364.650,168.838,52.477,160.003
C04331=1015.721,251.255,364.678,168.833,52.484,160.003
C04332=1015.715,251.007,364.705,168.828,52.491,160.004
C04333=1015.710,250.758,364.733,168.823,52.499,160.005
C04334=1015.704,250.510,364.760,168.819,52.507,160.006
C04335=1015.699,250.261,364.788,168.814,52.514,160.006
C04336=1015.693,250.013,364.815,168.809,52.522,160.007
C04337=1015.687,249.765,364.842,168.804,52.529,160.008
C04338=1015.682,249.527,364.868,168.800,52.536,160.008
C04339=1015.677,249.291,364.894,168.796,52.544,160.009
C04340=1015.672,249.053,364.921,168.791,52.551,160.010
C04341=1015.666,248.816,364.947,168.787,52.558,160.010
C04342=1015.661,248.578,364.973,168.781,52.565,160.011
C04343=1015.655,248.341,364.999,168.777,52.573,160.012
C04344=1015.651,248.104,365.025,168.772,52.580,160.012
C04345=1015.645,247.867,365.051,168.768,52.587,160.013
C04346=1015.640,247.619,365.079,168.763,52.595,160.014
C04347=1015.634,247.370,365.105,168.759,52.602,160.015
C04348=1015.629,247.122,365.133,168.754,52.610,160.015
C04349=1015.623,246.873,365.161,168.749,52.618,160.016
C04350=1015.618,246.625,365.187,168.744,52.625,160.017
C04351=1015.613,246.376,365.214,168.739,52.633,160.017
C04352=1015.606,246.128,365.242,168.735,52.640,160.018
C04353=1015.601,245.879,365.269,168.730,52.648,160.019
C04354=1015.596,245.631,365.297,168.725,52.656,160.020
C04355=1015.590,245.382,365.323,168.720,52.664,160.020
C04356=1015.585,245.134,365.351,168.715,52.671,160.021
C04357=1015.579,244.886,365.378,168.711,52.679,160.022
C04358=1015.574,244.637,365.405,168.706,52.687,160.023
C04359=1015.568,244.389,365.432,168.701,52.695,160.024
C04360=1015.563,244.140,365.459,168.696,52.703,160.024
C04361=1015.558,243.891,365.486,168.691,52.711,160.025
C04362=1015.552,243.644,365.514,168.687,52.718,160.026
C04363=1015.547,243.395,365.541,168.682,52.726,160.027
C04364=1015.541,243.147,365.568,168.678,52.734,160.027
C04365=1015.536,242.898,365.595,168.673,52.742,160.028
C04366=1015.530,242.650,365.621,168.668,52.750,160.029
C04367=1015.525,242.401,365.649,168.663,52.757,160.030
C04368=1015.520,242.153,365.675,168.659,52.766,160.031
C04369=1015.514,241.904,365.702,168.654,52.773,160.031
C04370=1015.509,241.656,365.729,168.650,52.781,160.032
C04371=1015.503,241.407,365.756,168.645,52.790,160.033
C04372=1015.497,241.159,365.782,168.640,52.797,160.034
C04373=1015.492,240.910,365.808,168.636,52.806,160.035
C04374=1015.487,240.661,365.836,168.631,52.814,160.035
C04375=1015.481,240.413,365.862,168.626,52.822,160.036
C04376=1015.475,240.165,365.889,168.621,52.830,160.037
C04377=1015.470,239.916,365.916,168.617,52.838,160.038
C04378=1015.464,239.667,365.943,168.612,52.846,160.039
C04379=1015.459,239.419,365.969,168.607,52.854,160.039
C04380=1015.454,239.170,365.996,168.602,52.862,160.040
C04381=1015.448,238.921,366.023,168.598,52.871,160.041
C04382=1015.442,238.673,366.049,168.593,52.879,160.042
C04383=1015.437,238.425,366.075,168.588,52.887,160.043
C04384=1015.432,238.176,366.102,168.583,52.895,160.044
C04385=1015.426,237.928,366.128,168.579,52.903,160.045
C04386=1015.420,237.679,366.154,168.574,52.912,160.045
C04387=1015.415,237.431,366.181,168.569,52.920,160.046
C04388=1015.409,237.182,366.207,168.565,52.928,160.047
C04389=1015.403,236.933,366.233,168.560,52.937,160.048
C04390=1015.398,236.685,366.260,168.556,52.945,160.049
C04391=1015.393,236.437,366.286,168.551,52.953,160.050
C04392=1015.387,236.188,366.312,168.546,52.961,160.051
C04393=1015.382,235.939,366.338,168.542,52.970,160.052
C04394=1015.376,235.691,366.365,168.537,52.978,160.053
C04395=1015.370,235.442,366.391,168.533,52.987,160.053
C04396=1015.365,235.194,366.417,168.528,52.995,160.054
C04397=1015.359,234.945,366.443,168.523,53.003,160.055
C04398=1015.354,234.705,366.468,168.519,53.012,160.056
C04399=1015.348,234.464,366.494,168.515,53.020,160.057
C04400=1015.344,234.223,366.520,168.510,53.028,160.058
C04401=1015.339,233.983,366.545,168.505,53.036,160.059
C04402=1015.333,233.742,366.570,168.501,53.045,160.060
C04403=1015.328,233.501,366.596,168.496,53.053,160.060
C04404=1015.323,233.262,366.621,168.492,53.061,160.061
C04405=1015.317,233.020,366.646,168.488,53.069,160.062
C04406=1015.311,232.772,366.672,168.483,53.078,160.063
C04407=1015.306,232.523,366.698,168.478,53.087,160.064
C04408=1015.301,232.275,366.724,168.473,53.095,160.065
C04409=1015.295,232.026,366.750,168.469,53.104,160.066
C04410=1015.290,231.777,366.776,168.464,53.112,160.067
C04411=1015.284,231.528,366.802,168.460,53.121,160.068
C04412=1015.278,231.281,366.828,168.455,53.129,160.069
C04413=1015.273,231.032,366.854,168.451,53.138,160.070
C04414=1015.268,230.783,366.880,168.446,53.147,160.070
C04415=1015.263,230.535,366.905,168.441,53.155,160.071
C04416=1015.257,230.286,366.932,168.437,53.164,160.072
C04417=1015.251,230.037,366.958,168.432,53.172,160.073
C04418=1015.247,229.789,366.983,168.428,53.181,160.074
C04419=1015.241,229.540,367.009,168.422,53.190,160.075
C04420=1015.236,229.291,367.035,168.418,53.199,160.076
C04421=1015.230,229.044,367.062,168.414,53.208,160.077
C04422=1015.224,228.795,367.087,168.409,53.216,160.078
C04423=1015.219,228.546,367.113,168.405,53.225,160.079
C04424=1015.214,228.298,367.138,168.400,53.234,160.080
C04425=1015.208,228.049,367.164,168.396,53.243,160.081
C04426=1015.203,227.800,367.190,168.391,53.251,160.082
C04427=1015.197,227.552,367.215,168.386,53.261,160.083
C04428=1015.192,227.303,367.241,168.382,53.270,160.084
C04429=1015.186,227.054,367.267,168.377,53.278,160.085
C04430=1015.182,226.805,367.293,168.373,53.287,160.086
C04431=1015.176,226.556,367.319,168.368,53.296,160.087
C04432=1015.171,226.309,367.344,168.363,53.305,160.088
C04433=1015.165,226.060,367.370,168.359,53.314,160.089
C04434=1015.160,225.811,367.396,168.354,53.323,160.090
C04435=1015.154,225.563,367.420,168.350,53.332,160.091
C04436=1015.149,225.314,367.446,168.346,53.341,160.092
C04437=1015.143,225.065,367.471,168.341,53.351,160.093
C04438=1015.138,224.816,367.497,168.336,53.359,160.094
C04439=1015.132,224.567,367.522,168.331,53.369,160.095
C04440=1015.127,224.319,367.547,168.327,53.378,160.096
C04441=1015.120,224.070,367.573,168.323,53.387,160.097
C04442=1015.116,223.822,367.598,168.318,53.396,160.098
C04443=1015.110,223.573,367.624,168.313,53.405,160.099
C04444=1015.105,223.325,367.649,168.309,53.415,160.100
C04445=1015.099,223.076,367.675,168.305,53.424,160.101
C04446=1015.094,222.827,367.699,168.300,53.432,160.102
C04447=1015.089,222.578,367.725,168.295,53.442,160.103
C04448=1015.083,222.330,367.750,168.291,53.451,160.104
C04449=1015.078,222.080,367.775,168.286,53.460,160.105
C04450=1015.072,221.832,367.800,168.282,53.470,160.106
C04451=1015.067,221.584,367.826,168.277,53.479,160.107
C04452=1015.061,221.335,367.850,168.273,53.488,160.109
C04453=1015.056,221.086,367.876,168.268,53.497,160.109
C04454=1015.050,220.838,367.901,168.264,53.507,160.111
C04455=1015.045,220.588,367.926,168.260,53.516,160.112
C04456=1015.040,220.340,367.952,168.255,53.526,160.113
C04457=1015.034,220.091,367.977,168.250,53.534,160.114
C04458=1015.029,219.847,368.001,168.246,53.544,160.115
C04459=1015.024,219.602,368.026,168.242,53.553,160.116
C04460=1015.018,219.357,368.051,168.238,53.563,160.117
C04461=1015.013,219.113,368.076,168.232,53.572,160.118
C04462=1015.008,218.867,368.101,168.228,53.581,160.119
C04463=1015.003,218.623,368.125,168.223,53.591,160.120
C04464=1014.998,218.379,368.150,168.219,53.599,160.121
C04465=1014.992,218.134,368.175,168.215,53.608,160.122
C04466=1014.987,217.885,368.199,168.210,53.618,160.123
C04467=1014.982,217.636,368.225,168.206,53.627,160.125
C04468=1014.976,217.388,368.249,168.201,53.637,160.126
C04469=1014.971,217.139,368.274,168.197,53.647,160.127
C04470=1014.965,216.890,368.299,168.193,53.656,160.128
C04471=1014.960,216.641,368.324,168.188,53.667,160.129
C04472=1014.955,216.393,368.348,168.183,53.676,160.130
C04473=1014.949,216.144,368.373,168.179,53.686,160.131
C04474=1014.943,215.896,368.398,168.175,53.695,160.132
C04475=1014.939,215.647,368.423,168.170,53.705,160.134
C04476=1014.933,215.398,368.448,168.166,53.714,160.135
C04477=1014.927,215.149,368.472,168.161,53.725,160.136
C04478=1014.922,214.901,368.496,168.156,53.734,160.137
C04479=1014.916,214.652,368.521,168.153,53.744,160.138
C04480=1014.911,214.403,368.547,168.148,53.754,160.139
C04481=1014.906,214.155,368.571,168.143,53.764,160.141
C04482=1014.900,213.905,368.596,168.139,53.773,160.142
C04483=1014.895,213.657,368.620,168.135,53.783,160.143
C04484=1014.890,213.408,368.645,168.130,53.793,160.144
C04485=1014.885,213.160,368.670,168.125,53.803,160.145
C04486=1014.879,212.911,368.694,168.121,53.812,160.146
C04487=1014.873,212.662,368.718,168.116,53.822,160.147
C04488=1014.869,212.413,368.743,168.112,53.833,160.149
C04489=1014.864,212.165,368.768,168.108,53.842,160.150
C04490=1014.858,211.915,368.792,168.103,53.852,160.151
C04491=1014.852,211.667,368.816,168.099,53.862,160.152
C04492=1014.847,211.419,368.841,168.094,53.872,160.153
C04493=1014.842,211.170,368.866,168.091,53.882,160.155
C04494=1014.836,210.921,368.891,168.086,53.892,160.156
C04495=1014.831,210.672,368.915,168.081,53.901,160.157
C04496=1014.826,210.423,368.939,168.077,53.912,160.158
C04497=1014.821,210.174,368.964,168.072,53.922,160.159
C04498=1014.816,209.926,368.989,168.068,53.932,160.161
C04499=1014.810,209.677,369.013,168.064,53.941,160.162
C04500=1014.805,209.428,369.037,168.059,53.952,160.163
C04501=1014.799,209.179,369.062,168.054,53.962,160.164
C04502=1014.794,208.931,369.086,168.050,53.972,160.165
C04503=1014.789,208.682,369.110,168.046,53.983,160.167
C04504=1014.783,208.434,369.134,168.042,53.992,160.168
C04505=1014.778,208.184,369.159,168.037,54.002,160.169
C04506=1014.772,207.936,369.183,168.033,54.013,160.170
C04507=1014.767,207.687,369.208,168.028,54.023,160.171
C04508=1014.762,207.438,369.231,168.024,54.033,160.173
C04509=1014.757,207.189,369.256,168.020,54.044,160.174
C04510=1014.752,206.940,369.280,168.015,54.053,160.175
C04511=1014.746,206.692,369.304,168.010,54.064,160.176
C04512=1014.741,206.444,369.328,168.006,54.074,160.178
C04513=1014.736,206.195,369.352,168.002,54.085,160.179
C04514=1014.731,205.946,369.376,167.997,54.095,160.180
C04515=1014.725,205.697,369.401,167.993,54.105,160.181
C04516=1014.719,205.448,369.425,167.988,54.116,160.183
C04517=1014.714,205.199,369.449,167.984,54.126,160.184
C04518=1014.709,204.968,369.471,167.980,54.136,160.185
C04519=1014.705,204.736,369.494,167.976,54.145,160.186
C04520=1014.699,204.503,369.516,167.972,54.155,160.188
C04521=1014.694,204.272,369.538,167.968,54.165,160.189
C04522=1014.689,204.039,369.560,167.963,54.175,160.190
C04523=1014.685,203.808,369.582,167.960,54.185,160.191
C04524=1014.680,203.576,369.605,167.955,54.195,160.192
C04525=1014.674,203.344,369.627,167.952,54.204,160.194
C04526=1014.655,202.228,369.727,167.429,54.129,160.062
C04527=1014.651,201.979,369.749,167.424,54.141,160.063
C04528=1014.646,201.730,369.771,167.419,54.153,160.064
C04529=1014.642,201.481,369.793,167.415,54.164,160.066
C04530=1014.638,201.232,369.815,167.410,54.176,160.067
C04531=1014.634,200.983,369.837,167.405,54.187,160.069
C04532=1014.630,200.734,369.860,167.400,54.199,160.070
C04533=1014.625,200.485,369.882,167.396,54.210,160.071
C04534=1014.621,200.236,369.904,167.391,54.222,160.073
C04535=1014.617,199.987,369.927,167.386,54.233,160.074
C04536=1014.612,199.738,369.948,167.382,54.245,160.075
C04537=1014.608,199.489,369.970,167.378,54.256,160.077
C04538=1014.605,199.240,369.992,167.373,54.268,160.078
C04539=1014.600,198.991,370.014,167.368,54.280,160.079
C04540=1014.596,198.742,370.037,167.363,54.291,160.081
C04541=1014.591,198.494,370.059,167.359,54.303,160.082
C04542=1014.587,198.244,370.080,167.354,54.314,160.084
C04543=1014.583,197.995,370.102,167.349,54.326,160.085
C04544=1014.578,197.745,370.123,167.344,54.338,160.086
C04545=1014.574,197.497,370.145,167.339,54.349,160.087
C04546=1014.570,197.248,370.167,167.335,54.361,160.089
C04547=1014.565,196.999,370.188,167.331,54.372,160.090
C04548=1014.560,196.750,370.210,167.326,54.384,160.092
C04549=1014.556,196.501,370.231,167.321,54.396,160.093
C04550=1014.552,196.252,370.253,167.316,54.408,160.094
C04551=1014.548,196.003,370.275,167.312,54.419,160.096
C04552=1014.543,195.754,370.296,167.308,54.431,160.097
C04553=1014.539,195.505,370.319,167.303,54.443,160.099
C04554=1014.535,195.256,370.340,167.298,54.454,160.100
C04555=1014.530,195.007,370.362,167.294,54.466,160.101
C04556=1014.526,194.758,370.383,167.289,54.477,160.103
C04557=1014.522,194.509,370.405,167.284,54.489,160.104
C04558=1014.518,194.260,370.426,167.279,54.501,160.105
C04559=1014.513,194.011,370.448,167.275,54.512,160.107
C04560=1014.508,193.762,370.469,167.271,54.524,160.108
C04561=1014.505,193.512,370.491,167.266,54.536,160.109
C04562=1014.500,193.264,370.512,167.262,54.548,160.111
C04563=1014.496,193.014,370.533,167.258,54.559,160.112
C04564=1014.492,192.765,370.556,167.253,54.571,160.114
C04565=1014.488,192.517,370.577,167.249,54.582,160.115
C04566=1014.483,192.268,370.598,167.244,54.594,160.117
C04567=1014.478,192.018,370.620,167.239,54.606,160.118
C04568=1014.475,191.769,370.641,167.235,54.617,160.119
C04569=1014.470,191.520,370.663,167.231,54.629,160.121
C04570=1014.466,191.271,370.684,167.226,54.641,160.122
C04571=1014.462,191.022,370.705,167.222,54.652,160.124
C04572=1014.458,190.773,370.727,167.217,54.664,160.125
C04573=1014.454,190.524,370.748,167.212,54.676,160.126
C04574=1014.450,190.275,370.769,167.208,54.687,160.128
C04575=1014.445,190.026,370.792,167.204,54.699,160.129
C04576=1014.442,189.777,370.812,167.199,54.710,160.130
C04577=1014.437,189.528,370.834,167.195,54.722,160.132
C04578=1014.433,189.280,370.855,167.190,54.734,160.133
C04579=1014.429,189.030,370.877,167.186,54.745,160.135
C04580=1014.424,188.780,370.898,167.182,54.757,160.136
C04581=1014.420,188.532,370.919,167.178,54.768,160.137
C04582=1014.416,188.283,370.941,167.173,54.780,160.139
C04583=1014.413,188.034,370.962,167.168,54.792,160.140
C04584=1014.408,187.784,370.983,167.164,54.803,160.141
C04585=1014.404,187.536,371.004,167.160,54.815,160.143
C04586=1014.400,187.286,371.026,167.156,54.826,160.144
C04587=1014.396,187.007,371.050,167.151,54.840,160.146
C04588=1014.391,186.727,371.074,167.146,54.853,160.147
C04589=1014.386,186.448,371.098,167.142,54.865,160.149
C04590=1014.382,186.169,371.121,167.137,54.879,160.151
C04591=1014.377,185.920,371.143,167.133,54.890,160.152
C04592=1014.373,185.671,371.164,167.128,54.902,160.154
C04593=1014.369,185.422,371.185,167.125,54.913,160.155
C04594=1014.366,185.173,371.206,167.120,54.925,160.156
C04595=1014.361,184.923,371.227,167.116,54.937,160.158
C04596=1014.357,184.675,371.248,167.111,54.948,160.159
C04597=1014.353,184.425,371.269,167.108,54.960,160.161
C04598=1014.350,184.176,371.291,167.103,54.972,160.162
C04599=1014.345,183.927,371.313,167.099,54.983,160.163
C04600=1014.341,183.679,371.333,167.094,54.995,160.165
C04601=1014.336,183.429,371.355,167.090,55.006,160.166
C04602=1014.333,183.180,371.376,167.085,55.018,160.167
C04603=1014.329,182.931,371.397,167.082,55.029,160.169
C04604=1014.325,182.682,371.418,167.078,55.040,160.170
C04605=1014.321,182.433,371.439,167.073,55.052,160.172
C04606=1014.317,182.183,371.460,167.070,55.064,160.173
C04607=1014.313,181.935,371.481,167.065,55.075,160.174
C04608=1014.309,181.685,371.502,167.061,55.087,160.176
C04609=1014.305,181.437,371.523,167.057,55.098,160.177
C04610=1014.300,181.186,371.544,167.053,55.110,160.179
C04611=1014.296,180.938,371.564,167.049,55.123,160.180
C04612=1014.292,180.689,371.585,167.045,55.134,160.182
C04613=1014.288,180.439,371.605,167.040,55.146,160.183
C04614=1014.283,180.191,371.625,167.037,55.158,160.185
C04615=1014.279,179.941,371.646,167.032,55.170,160.186
C04616=1014.275,179.692,371.666,167.028,55.182,160.188
C04617=1014.270,179.444,371.687,167.024,55.193,160.189
C04618=1014.266,179.194,371.707,167.019,55.205,160.190
C04619=1014.261,178.945,371.727,167.016,55.217,160.192
C04620=1014.257,178.695,371.748,167.011,55.229,160.194
C04621=1014.253,178.446,371.768,167.008,55.241,160.195
C04622=1014.249,178.198,371.789,167.003,55.253,160.196
C04623=1014.244,177.948,371.809,167.000,55.264,160.198
C04624=1014.240,177.699,371.829,166.995,55.276,160.199
C04625=1014.236,177.450,371.849,166.992,55.288,160.201
C04626=1014.232,177.201,371.870,166.987,55.300,160.202
C04627=1014.227,176.952,371.890,166.983,55.312,160.204
C04628=1014.223,176.703,371.911,166.979,55.324,160.205
C04629=1014.218,176.453,371.930,166.975,55.335,160.207
C04630=1014.214,176.204,371.951,166.971,55.348,160.208
C04631=1014.211,175.955,371.971,166.967,55.359,160.210
C04632=1014.206,175.706,371.992,166.963,55.371,160.211
C04633=1014.202,175.457,372.012,166.959,55.383,160.213
C04634=1014.197,175.208,372.032,166.955,55.394,160.214
C04635=1014.194,174.959,372.052,166.951,55.406,160.215
C04636=1014.189,174.709,372.073,166.946,55.418,160.217
C04637=1014.185,174.460,372.093,166.943,55.430,160.218
C04638=1014.181,174.211,372.113,166.939,55.442,160.220
C04639=1014.177,173.963,372.133,166.935,55.453,160.221
C04640=1014.172,173.713,372.154,166.931,55.465,160.223
C04641=1014.168,173.464,372.174,166.927,55.477,160.224
C04642=1014.164,173.215,372.194,166.923,55.488,160.226
C04643=1014.160,172.965,372.214,166.919,55.500,160.227
C04644=1014.155,172.716,372.234,166.915,55.512,160.229
C04645=1014.152,172.467,372.254,166.912,55.524,160.230
C04646=1014.148,172.218,372.275,166.907,55.536,160.232
C04647=1014.143,171.969,372.295,166.904,55.548,160.233
C04648=1014.140,171.720,372.315,166.900,55.559,160.235
C04649=1014.134,171.471,372.335,166.896,55.571,160.236
C04650=1014.131,171.221,372.355,166.892,55.583,160.238
C04651=1014.126,170.942,372.378,166.887,55.596,160.239
C04652=1014.121,170.662,372.400,166.884,55.609,160.241
C04653=1014.117,170.382,372.423,166.879,55.622,160.242
C04654=1014.113,170.103,372.445,166.875,55.636,160.244
C04655=1014.109,169.854,372.466,166.871,55.647,160.246
C04656=1014.104,169.605,372.485,166.867,55.659,160.247
C04657=1014.101,169.356,372.505,166.863,55.671,160.249
C04658=1014.096,169.107,372.526,166.860,55.682,160.250
C04659=1014.092,168.858,372.546,166.855,55.694,160.251
C04660=1014.087,168.608,372.566,166.852,55.706,160.253
C04661=1014.084,168.359,372.586,166.848,55.717,160.254
C04662=1014.080,168.109,372.606,166.845,55.729,160.256
C04663=1014.076,167.861,372.626,166.840,55.741,160.257
C04664=1014.072,167.612,372.646,166.837,55.752,160.259
C04665=1014.068,167.363,372.665,166.833,55.764,160.260
C04666=1014.064,167.113,372.685,166.830,55.776,160.262
C04667=1014.060,166.864,372.706,166.825,55.788,160.263
C04668=1014.056,166.616,372.726,166.822,55.799,160.265
C04669=1014.052,166.366,372.746,166.818,55.811,160.266
C04670=1014.047,166.116,372.766,166.815,55.822,160.268
C04671=1014.044,165.867,372.786,166.811,55.834,160.269
C04672=1014.039,165.618,372.805,166.807,55.846,160.271
C04673=1014.036,165.369,372.825,166.803,55.858,160.272
C04674=1014.032,165.120,372.846,166.800,55.869,160.274
C04675=1014.027,164.871,372.866,166.796,55.881,160.275
C04676=1014.024,164.622,372.886,166.793,55.892,160.277
C04677=1014.019,164.372,372.905,166.788,55.904,160.278
C04678=1014.016,164.123,372.925,166.785,55.916,160.280
C04679=1014.011,163.874,372.945,166.782,55.928,160.281
C04680=1014.008,163.625,372.965,166.778,55.938,160.282
C04681=1014.004,163.375,372.985,166.774,55.950,160.284
C04682=1014.000,163.126,373.004,166.771,55.962,160.285
C04683=1013.996,162.877,373.024,166.767,55.973,160.287
C04684=1013.992,162.629,373.044,166.764,55.985,160.288
C04685=1013.988,162.379,373.065,166.759,55.997,160.290
C04686=1013.984,162.130,373.085,166.756,56.009,160.291
C04687=1013.980,161.881,373.104,166.752,56.020,160.293
C04688=1013.976,161.631,373.124,166.749,56.032,160.294
C04689=1013.972,161.382,373.144,166.746,56.043,160.296
C04690=1013.968,161.133,373.164,166.742,56.054,160.297
C04691=1013.964,160.884,373.183,166.738,56.066,160.299
C04692=1013.960,160.635,373.203,166.735,56.078,160.300
C04693=1013.957,160.385,373.223,166.731,56.089,160.302
C04694=1013.953,160.136,373.243,166.728,56.101,160.303
C04695=1013.950,159.888,373.262,166.725,56.113,160.305
C04696=1013.945,159.639,373.282,166.721,56.124,160.306
C04697=1013.942,159.389,373.302,166.717,56.135,160.308
C04698=1013.937,159.140,373.321,166.714,56.147,160.309
C04699=1013.934,158.890,373.341,166.711,56.158,160.311
C04700=1013.930,158.641,373.361,166.707,56.170,160.312
C04701=1013.926,158.392,373.380,166.703,56.181,160.314
C04702=1013.922,158.142,373.400,166.700,56.193,160.315
C04703=1013.918,157.893,373.420,166.696,56.204,160.317
C04704=1013.914,157.644,373.439,166.692,56.216,160.318
C04705=1013.910,157.395,373.458,166.689,56.228,160.319
C04706=1013.905,157.146,373.478,166.685,56.240,160.321
C04707=1013.901,156.896,373.496,166.682,56.252,160.323
C04708=1013.897,156.647,373.516,166.679,56.263,160.324
C04709=1013.893,156.398,373.535,166.675,56.275,160.326
C04710=1013.889,156.148,373.555,166.672,56.287,160.327
C04711=1013.885,155.900,373.574,166.669,56.298,160.329
C04712=1013.881,155.650,373.592,166.664,56.310,160.330
C04713=1013.877,155.401,373.612,166.661,56.322,160.332
C04714=1013.873,155.152,373.631,166.657,56.334,160.333
C04715=1013.868,154.872,373.653,166.654,56.347,160.335
C04716=1013.863,154.592,373.674,166.650,56.360,160.337
C04717=1013.859,154.312,373.695,166.647,56.373,160.338
C04718=1013.855,154.032,373.717,166.643,56.386,160.340
C04719=1013.850,153.783,373.736,166.639,56.397,160.342
C04720=1013.846,153.534,373.756,166.635,56.410,160.343
C04721=1013.842,153.284,373.774,166.632,56.421,160.345
C04722=1013.838,153.036,373.794,166.628,56.433,160.346
C04723=1013.834,152.786,373.812,166.625,56.445,160.348
C04724=1013.831,152.537,373.832,166.622,56.456,160.349
C04725=1013.827,152.287,373.851,166.619,56.468,160.351
C04726=1013.823,152.038,373.870,166.615,56.480,160.352
C04727=1013.817,151.789,373.889,166.611,56.491,160.354
C04728=1013.814,151.540,373.907,166.608,56.503,160.355
C04729=1013.810,151.291,373.927,166.605,56.514,160.357
C04730=1013.806,151.041,373.945,166.602,56.526,160.358
C04731=1013.801,150.792,373.965,166.598,56.538,160.360
C04732=1013.798,150.543,373.983,166.595,56.549,160.361
C04733=1013.794,150.294,374.002,166.592,56.561,160.363
C04734=1013.789,150.045,374.021,166.589,56.573,160.365
C04735=1013.785,149.795,374.040,166.585,56.585,160.366
C04736=1013.781,149.545,374.059,166.582,56.596,160.368
C04737=1013.778,149.297,374.078,166.578,56.607,160.369
C04738=1013.774,149.047,374.097,166.575,56.619,160.370
C04739=1013.770,148.798,374.116,166.572,56.631,160.372
C04740=1013.765,148.549,374.135,166.568,56.643,160.374
C04741=1013.762,148.300,374.153,166.565,56.654,160.375
C04742=1013.758,148.050,374.172,166.563,56.666,160.377
C04743=1013.753,147.801,374.191,166.559,56.677,160.378
C04744=1013.749,147.552,374.209,166.556,56.688,160.380
C04745=1013.745,147.303,374.228,166.553,56.700,160.381
C04746=1013.741,147.053,374.247,166.550,56.712,160.383
C04747=1013.737,146.804,374.266,166.546,56.724,160.384
C04748=1013.733,146.555,374.285,166.543,56.736,160.386
C04749=1013.729,146.305,374.304,166.539,56.747,160.387
C04750=1013.724,146.056,374.322,166.536,56.758,160.389
C04751=1013.721,145.808,374.341,166.533,56.770,160.390
C04752=1013.717,145.558,374.360,166.530,56.782,160.392
C04753=1013.713,145.308,374.378,166.526,56.794,160.394
C04754=1013.709,145.059,374.397,166.524,56.804,160.395
C04755=1013.704,144.810,374.415,166.521,56.816,160.397
C04756=1013.700,144.560,374.434,166.517,56.828,160.398
C04757=1013.697,144.311,374.452,166.514,56.840,160.400
C04758=1013.692,144.062,374.470,166.511,56.851,160.401
C04759=1013.688,143.812,374.489,166.508,56.863,160.403
C04760=1013.685,143.563,374.507,166.504,56.874,160.404
C04761=1013.680,143.314,374.526,166.501,56.886,160.406
C04762=1013.676,143.065,374.545,166.498,56.898,160.407
C04763=1013.672,142.816,374.563,166.495,56.910,160.409
C04764=1013.667,142.567,374.582,166.491,56.921,160.411
C04765=1013.663,142.317,374.600,166.489,56.932,160.412
C04766=1013.660,142.068,374.619,166.486,56.944,160.414
C04767=1013.655,141.819,374.637,166.482,56.956,160.415
C04768=1013.651,141.569,374.656,166.479,56.968,160.417
C04769=1013.648,141.320,374.674,166.476,56.979,160.418
C04770=1013.643,141.071,374.692,166.472,56.990,160.420
C04771=1013.639,140.822,374.711,166.469,57.002,160.421
C04772=1013.635,140.572,374.729,166.467,57.014,160.423
C04773=1013.631,140.323,374.748,166.463,57.025,160.424
C04774=1013.627,140.073,374.765,166.460,57.037,160.426
C04775=1013.623,139.824,374.783,166.457,57.048,160.427
C04776=1013.619,139.575,374.802,166.454,57.060,160.429
C04777=1013.615,139.325,374.820,166.451,57.071,160.431
C04778=1013.611,139.077,374.838,166.448,57.083,160.432
C04779=1013.606,138.796,374.860,166.445,57.096,160.434
C04780=1013.602,138.517,374.880,166.441,57.109,160.436
C04781=1013.597,138.237,374.901,166.438,57.122,160.437
C04782=1013.593,137.957,374.921,166.435,57.134,160.439
C04783=1013.589,137.707,374.939,166.431,57.145,160.440
C04784=1013.585,137.458,374.958,166.428,57.157,160.442
C04785=1013.580,137.209,374.976,166.425,57.169,160.444
C04786=1013.577,136.960,374.994,166.423,57.180,160.445
C04787=1013.573,136.710,375.012,166.419,57.192,160.447
C04788=1013.569,136.461,375.030,166.416,57.203,160.448
C04789=1013.564,136.212,375.048,166.413,57.215,160.450
C04790=1013.560,135.963,375.066,166.411,57.226,160.451
C04791=1013.556,135.713,375.085,166.408,57.238,160.453
C04792=1013.552,135.464,375.102,166.404,57.249,160.454
C04793=1013.548,135.215,375.121,166.401,57.261,160.456
C04794=1013.544,134.966,375.139,166.399,57.272,160.458
C04795=1013.540,134.716,375.157,166.395,57.283,160.459
C04796=1013.536,134.467,375.174,166.392,57.295,160.461
C04797=1013.532,134.217,375.193,166.390,57.307,160.462
C04798=1013.528,133.968,375.210,166.387,57.318,160.464
C04799=1013.523,133.719,375.228,166.384,57.330,160.465
C04800=1013.520,133.470,375.247,166.380,57.341,160.467
C04801=1013.515,133.220,375.264,166.378,57.352,160.468
C04802=1013.511,132.971,375.282,166.375,57.364,160.470
C04803=1013.507,132.721,375.301,166.371,57.375,160.471
C04804=1013.503,132.472,375.318,166.369,57.387,160.473
C04805=1013.499,132.222,375.337,166.366,57.398,160.474
C04806=1013.495,131.973,375.354,166.363,57.410,160.476
C04807=1013.491,131.724,375.372,166.360,57.421,160.478
C04808=1013.487,131.475,375.390,166.357,57.432,160.479
C04809=1013.483,131.225,375.408,166.355,57.443,160.481
C04810=1013.479,130.976,375.425,166.352,57.455,160.482
C04811=1013.475,130.727,375.443,166.348,57.466,160.484
C04812=1013.471,130.477,375.461,166.346,57.478,160.485
C04813=1013.467,130.228,375.480,166.343,57.489,160.487
C04814=1013.463,129.978,375.497,166.341,57.500,160.489
C04815=1013.459,129.730,375.515,166.337,57.512,160.490
C04816=1013.455,129.479,375.533,166.334,57.523,160.491
C04817=1013.451,129.231,375.551,166.332,57.534,160.493
C04818=1013.446,128.981,375.568,166.329,57.546,160.495
C04819=1013.442,128.732,375.585,166.325,57.557,160.496
C04820=1013.438,128.483,375.603,166.323,57.569,160.498
C04821=1013.434,128.233,375.621,166.320,57.581,160.499
C04822=1013.430,127.984,375.638,166.317,57.592,160.501
C04823=1013.425,127.734,375.656,166.315,57.603,160.503
C04824=1013.421,127.485,375.673,166.311,57.615,160.504
C04825=1013.417,127.236,375.690,166.309,57.626,160.506
C04826=1013.412,126.986,375.708,166.306,57.637,160.507
C04827=1013.409,126.737,375.725,166.303,57.649,160.509
C04828=1013.405,126.488,375.742,166.300,57.660,160.510
C04829=1013.400,126.239,375.760,166.297,57.672,160.512
C04830=1013.396,125.989,375.777,166.295,57.683,160.513
C04831=1013.392,125.739,375.795,166.292,57.695,160.515
C04832=1013.388,125.490,375.812,166.288,57.706,160.516
C04833=1013.384,125.241,375.830,166.286,57.717,160.518
C04834=1013.380,124.991,375.848,166.283,57.729,160.519
C04835=1013.376,124.742,375.865,166.281,57.740,160.521
C04836=1013.372,124.493,375.882,166.278,57.751,160.523
C04837=1013.367,124.243,375.900,166.276,57.763,160.524
C04838=1013.363,123.994,375.917,166.272,57.774,160.526
C04839=1013.360,123.745,375.934,166.270,57.785,160.527
C04840=1013.355,123.495,375.952,166.267,57.797,160.529
C04841=1013.351,123.246,375.970,166.264,57.808,160.530
C04842=1013.347,122.997,375.987,166.262,57.820,160.532
C04843=1013.342,122.717,376.006,166.259,57.832,160.534
C04844=1013.338,122.437,376.025,166.255,57.845,160.536
C04845=1013.333,122.158,376.044,166.252,57.857,160.537
C04846=1013.329,121.878,376.064,166.249,57.870,160.539
C04847=1013.324,121.628,376.082,166.247,57.881,160.540
C04848=1013.320,121.378,376.099,166.243,57.892,160.542
C04849=1013.316,121.129,376.116,166.241,57.903,160.544
C04850=1013.312,120.881,376.134,166.238,57.915,160.545
C04851=1013.308,120.631,376.151,166.236,57.925,160.547
C04852=1013.304,120.381,376.168,166.234,57.937,160.548
C04853=1013.300,120.132,376.185,166.230,57.948,160.550
C04854=1013.296,119.883,376.202,166.228,57.959,160.551
C04855=1013.292,119.633,376.220,166.224,57.970,160.553
C04856=1013.288,119.384,376.237,166.222,57.981,160.554
C04857=1013.284,119.135,376.255,166.220,57.993,160.556
C04858=1013.280,118.886,376.272,166.217,58.004,160.557
C04859=1013.275,118.636,376.289,166.214,58.015,160.559
C04860=1013.271,118.386,376.306,166.212,58.026,160.560
C04861=1013.268,118.137,376.323,166.209,58.037,160.562
C04862=1013.264,117.888,376.340,166.206,58.048,160.563
C04863=1013.259,117.638,376.358,166.205,58.059,160.565
C04864=1013.255,117.389,376.375,166.202,58.070,160.567
C04865=1013.251,117.139,376.392,166.199,58.081,160.568
C04866=1013.248,116.890,376.409,166.196,58.092,160.570
C04867=1013.243,116.641,376.427,166.194,58.103,160.571
C04868=1013.239,116.391,376.444,166.191,58.114,160.573
C04869=1013.235,116.142,376.461,166.188,58.125,160.574
C04870=1013.231,115.893,376.479,166.186,58.136,160.576
C04871=1013.227,115.644,376.496,166.184,58.147,160.577
C04872=1013.223,115.394,376.513,166.181,58.158,160.579
C04873=1013.219,115.144,376.530,166.178,58.169,160.580
C04874=1013.215,114.895,376.547,166.175,58.180,160.582
C04875=1013.211,114.646,376.564,166.173,58.191,160.583
C04876=1013.207,114.397,376.581,166.171,58.202,160.585
C04877=1013.203,114.147,376.598,166.168,58.212,160.586
C04878=1013.199,113.897,376.616,166.165,58.224,160.588
C04879=1013.195,113.648,376.633,166.163,58.235,160.589
C04880=1013.191,113.399,376.650,166.160,58.245,160.591
C04881=1013.187,113.150,376.667,166.158,58.256,160.592
C04882=1013.183,112.900,376.684,166.156,58.267,160.594
C04883=1013.180,112.651,376.701,166.154,58.278,160.596
C04884=1013.176,112.402,376.718,166.151,58.288,160.597
C04885=1013.171,112.152,376.736,166.147,58.300,160.598
C04886=1013.167,111.902,376.753,166.145,58.310,160.600
C04887=1013.164,111.653,376.770,166.143,58.321,160.601
C04888=1013.160,111.404,376.787,166.140,58.332,160.603
C04889=1013.155,111.154,376.803,166.138,58.343,160.604
C04890=1013.151,110.905,376.820,166.136,58.354,160.606
C04891=1013.148,110.656,376.837,166.134,58.365,160.608
C04892=1013.142,110.406,376.854,166.130,58.376,160.609
C04893=1013.139,110.156,376.870,166.128,58.387,160.611
C04894=1013.135,109.907,376.887,166.126,58.398,160.612
C04895=1013.131,109.658,376.904,166.123,58.409,160.614
C04896=1013.126,109.409,376.921,166.120,58.419,160.615
C04897=1013.123,109.159,376.937,166.118,58.430,160.617
C04898=1013.119,108.910,376.954,166.116,58.441,160.618
C04899=1013.114,108.661,376.971,166.114,58.452,160.620
C04900=1013.111,108.411,376.987,166.110,58.463,160.621
C04901=1013.106,108.162,377.004,166.108,58.474,160.623
C04902=1013.102,107.912,377.021,166.106,58.485,160.624
C04903=1013.097,107.662,377.037,166.104,58.496,160.626
C04904=1013.094,107.413,377.054,166.101,58.507,160.627
C04905=1013.089,107.164,377.070,166.099,58.517,160.629
C04906=1013.085,106.914,377.087,166.096,58.528,160.630
C04907=1013.081,106.635,377.105,166.094,58.540,160.632
C04908=1013.076,106.355,377.124,166.091,58.552,160.634
C04909=1013.071,106.076,377.142,166.088,58.564,160.635
C04910=1013.067,105.796,377.161,166.086,58.576,160.637
C04911=1013.063,105.547,377.178,166.082,58.587,160.639
C04912=1013.058,105.297,377.193,166.080,58.598,160.640
C04913=1013.055,105.048,377.210,166.078,58.609,160.642
C04914=1013.050,104.798,377.226,166.075,58.619,160.643
C04915=1013.046,104.549,377.243,166.073,58.630,160.645
C04916=1013.042,104.300,377.259,166.071,58.641,160.646
C04917=1013.038,104.050,377.276,166.068,58.651,160.647
C04918=1013.034,103.801,377.293,166.066,58.662,160.649
C04919=1013.030,103.552,377.309,166.065,58.673,160.651
C04920=1013.025,103.303,377.326,166.062,58.683,160.652
C04921=1013.022,103.053,377.342,166.060,58.694,160.654
C04922=1013.017,102.804,377.358,166.057,58.705,160.655
C04923=1013.014,102.554,377.375,166.055,58.715,160.657
C04924=1013.009,102.305,377.391,166.052,58.726,160.658
C04925=1013.006,102.055,377.408,166.050,58.736,160.659
C04926=1013.001,101.806,377.424,166.047,58.747,160.661
C04927=1012.997,101.556,377.440,166.045,58.758,160.663
C04928=1012.993,101.307,377.457,166.042,58.768,160.664
C04929=1012.989,101.057,377.473,166.040,58.779,160.666
C04930=1012.985,100.808,377.490,166.039,58.789,160.667
C04931=1012.981,100.558,377.506,166.036,58.800,160.669
C04932=1012.977,100.309,377.522,166.034,58.810,160.670
C04933=1012.973,100.060,377.539,166.031,58.821,160.672
C04934=1012.969,99.810,377.555,166.029,58.831,160.673
C04935=1012.965,99.561,377.572,166.027,58.842,160.674
C04936=1012.961,99.311,377.588,166.025,58.852,160.676
C04937=1012.956,99.062,377.605,166.022,58.862,160.677
C04938=1012.953,98.812,377.621,166.020,58.873,160.679
C04939=1012.949,98.562,377.637,166.017,58.884,160.680
C04940=1012.944,98.313,377.653,166.015,58.895,160.682
C04941=1012.940,98.064,377.669,166.013,58.904,160.683
C04942=1012.936,97.814,377.685,166.011,58.915,160.685
C04943=1012.932,97.564,377.701,166.008,58.926,160.686
C04944=1012.927,97.315,377.718,166.006,58.936,160.688
C04945=1012.923,97.066,377.733,166.004,58.947,160.689
C04946=1012.919,96.816,377.749,166.003,58.957,160.691
C04947=1012.916,96.567,377.765,166.000,58.967,160.692
C04948=1012.911,96.318,377.782,165.997,58.978,160.694
C04949=1012.907,96.069,377.797,165.995,58.989,160.695
C04950=1012.902,95.819,377.813,165.992,58.999,160.696
C04951=1012.898,95.569,377.829,165.991,59.009,160.698
C04952=1012.894,95.320,377.845,165.988,59.020,160.700
C04953=1012.890,95.071,377.862,165.986,59.030,160.701
C04954=1012.886,94.821,377.878,165.984,59.041,160.703
C04955=1012.881,94.571,377.893,165.982,59.051,160.704
C04956=1012.878,94.322,377.910,165.979,59.061,160.705
C04957=1012.874,94.073,377.925,165.977,59.071,160.707
C04958=1012.870,93.823,377.941,165.976,59.082,160.708
C04959=1012.865,93.574,377.957,165.973,59.092,160.710
C04960=1012.861,93.325,377.973,165.970,59.102,160.711
C04961=1012.857,93.075,377.990,165.969,59.112,160.713
C04962=1012.853,92.825,378.005,165.966,59.123,160.714
C04963=1012.849,92.576,378.021,165.965,59.133,160.716
C04964=1012.844,92.326,378.037,165.962,59.143,160.717
C04965=1012.840,92.078,378.053,165.959,59.153,160.718
C04966=1012.837,91.828,378.069,165.958,59.163,160.720
C04967=1012.832,91.578,378.085,165.955,59.174,160.721
C04968=1012.828,91.329,378.101,165.954,59.184,160.723
C04969=1012.824,91.079,378.117,165.951,59.194,160.724
C04970=1012.819,90.829,378.132,165.949,59.205,160.726
C04971=1012.816,90.594,378.147,165.946,59.214,160.727
C04972=1012.812,90.359,378.163,165.945,59.224,160.728
C04973=1012.808,90.124,378.177,165.943,59.233,160.730
C04974=1012.805,89.889,378.193,165.941,59.242,160.731
C04975=1012.800,89.654,378.208,165.939,59.252,160.732
C04976=1012.797,89.418,378.222,165.937,59.261,160.734
C04977=1012.793,89.183,378.237,165.935,59.270,160.735
C04978=1012.789,88.948,378.253,165.933,59.280,160.737
C04979=1012.785,88.699,378.268,165.931,59.291,160.738
C04980=1012.781,88.449,378.284,165.929,59.300,160.739
C04981=1012.776,88.200,378.300,165.926,59.311,160.741
C04982=1012.772,87.950,378.316,165.925,59.321,160.742
C04983=1012.769,87.701,378.330,165.922,59.331,160.744
C04984=1012.764,87.451,378.346,165.921,59.341,160.745
C04985=1012.760,87.202,378.362,165.918,59.351,160.746
C04986=1012.756,86.952,378.378,165.916,59.361,160.748
C04987=1012.752,86.703,378.393,165.914,59.371,160.749
C04988=1012.747,86.454,378.408,165.912,59.381,160.751
C04989=1012.743,86.204,378.424,165.911,59.391,160.752
C04990=1012.739,85.954,378.439,165.908,59.401,160.754
C04991=1012.734,85.704,378.455,165.906,59.411,160.755
C04992=1012.731,85.456,378.470,165.904,59.421,160.757
C04993=1012.726,85.206,378.486,165.902,59.430,160.758
C04994=1012.722,84.956,378.502,165.899,59.441,160.759
C04995=1012.718,84.707,378.518,165.897,59.451,160.761
C04996=1012.714,84.457,378.532,165.896,59.460,160.762
C04997=1012.709,84.208,378.547,165.893,59.471,160.764
C04998=1012.705,83.959,378.563,165.892,59.481,160.765
C04999=1012.676,96.231,377.382,165.960,59.184,160.725
C05000=1012.680,96.481,377.366,165.963,59.174,160.724
C05001=1012.685,96.730,377.350,165.965,59.164,160.722
C05002=1012.688,96.979,377.334,165.967,59.154,160.721
C05003=1012.692,97.229,377.318,165.969,59.143,160.719
C05004=1012.697,97.478,377.302,165.971,59.133,160.718
C05005=1012.701,97.728,377.287,165.974,59.123,160.716
C05006=1012.705,97.977,377.271,165.976,59.113,160.715
C05007=1012.709,98.227,377.254,165.979,59.102,160.713
C05008=1012.713,98.476,377.238,165.980,59.092,160.712
C05009=1012.718,98.726,377.222,165.983,59.082,160.711
C05010=1012.721,98.976,377.206,165.985,59.071,160.709
C05011=1012.726,99.225,377.189,165.987,59.061,160.707
C05012=1012.729,99.474,377.173,165.989,59.051,160.706
C05013=1012.733,99.723,377.158,165.992,59.040,160.705
C05014=1012.737,99.973,377.140,165.993,59.030,160.703
C05015=1012.741,100.222,377.125,165.996,59.020,160.702
C05016=1012.745,100.472,377.108,165.999,59.009,160.700
C05017=1012.749,100.721,377.092,166.000,59.000,160.699
C05018=1012.753,100.971,377.075,166.002,58.989,160.697
C05019=1012.758,101.220,377.059,166.005,58.978,160.696
C05020=1012.761,101.470,377.043,166.008,58.968,160.695
C05021=1012.766,101.719,377.026,166.009,58.958,160.693
C05022=1012.769,101.969,377.010,166.012,58.947,160.692
C05023=1012.774,102.218,376.994,166.014,58.936,160.690
C05024=1012.777,102.467,376.977,166.016,58.926,160.689
C05025=1012.781,102.716,376.962,166.019,58.916,160.687
C05026=1012.785,102.966,376.944,166.020,58.905,160.686
C05027=1012.789,103.215,376.929,166.023,58.895,160.684
C05028=1012.793,103.465,376.912,166.025,58.884,160.683
C05029=1012.798,103.714,376.896,166.028,58.874,160.681
C05030=1012.801,103.963,376.879,166.030,58.863,160.680
C05031=1012.806,104.213,376.863,166.033,58.853,160.678
C05032=1012.809,104.463,376.847,166.035,58.842,160.677
C05033=1012.814,104.712,376.830,166.038,58.832,160.676
C05034=1012.818,104.962,376.814,166.039,58.821,160.674
C05035=1012.821,105.211,376.797,166.041,58.810,160.672
C05036=1012.828,105.628,376.769,166.046,58.792,160.670
C05037=1012.835,106.045,376.742,166.049,58.774,160.667
C05038=1012.842,106.462,376.714,166.053,58.757,160.665
C05039=1012.849,106.879,376.687,166.058,58.739,160.662
C05040=1012.853,107.130,376.671,166.060,58.728,160.661
C05041=1012.857,107.379,376.654,166.063,58.718,160.659
C05042=1012.862,107.629,376.638,166.065,58.707,160.658
C05043=1012.865,107.878,376.621,166.067,58.696,160.656
C05044=1012.870,108.127,376.605,166.069,58.685,160.655
C05045=1012.874,108.377,376.588,166.072,58.675,160.653
C05046=1012.878,108.626,376.572,166.074,58.664,160.652
C05047=1012.882,108.876,376.555,166.076,58.653,160.650
C05048=1012.886,109.125,376.538,166.079,58.642,160.649
C05049=1012.890,109.374,376.522,166.081,58.632,160.647
C05050=1012.894,109.624,376.505,166.084,58.621,160.646
C05051=1012.898,109.873,376.488,166.086,58.610,160.644
C05052=1012.902,110.122,376.472,166.089,58.600,160.643
C05053=1012.906,110.372,376.455,166.091,58.589,160.641
C05054=1012.910,110.621,376.438,166.093,58.578,160.640
C05055=1012.914,110.870,376.422,166.095,58.567,160.638
C05056=1012.918,111.120,376.405,166.098,58.556,160.636
C05057=1012.922,111.369,376.388,166.101,58.545,160.635
C05058=1012.926,111.618,376.371,166.104,58.534,160.634
C05059=1012.930,111.867,376.355,166.106,58.524,160.632
C05060=1012.935,112.118,376.338,166.108,58.513,160.631
C05061=1012.938,112.368,376.320,166.110,58.502,160.629
C05062=1012.942,112.617,376.303,166.113,58.492,160.628
C05063=1012.945,112.866,376.286,166.116,58.481,160.626
C05064=1012.949,113.115,376.269,166.118,58.470,160.625
C05065=1012.953,113.365,376.252,166.120,58.459,160.623
C05066=1012.957,113.614,376.235,166.123,58.449,160.622
C05067=1012.961,113.863,376.218,166.125,58.438,160.620
C05068=1012.965,114.112,376.201,166.127,58.427,160.619
C05069=1012.969,114.362,376.184,166.130,58.416,160.617
C05070=1012.973,114.612,376.166,166.133,58.405,160.616
C05071=1012.977,114.861,376.149,166.135,58.394,160.614
C05072=1012.981,115.110,376.132,166.138,58.384,160.613
C05073=1012.985,115.359,376.115,166.140,58.373,160.611
C05074=1012.989,115.609,376.098,166.143,58.362,160.610
C05075=1012.992,115.858,376.081,166.145,58.351,160.608
C05076=1012.996,116.108,376.064,166.147,58.340,160.607
C05077=1013.000,116.357,376.047,166.151,58.329,160.605
C05078=1013.004,116.607,376.030,166.153,58.318,160.604
C05079=1013.008,116.856,376.013,166.155,58.307,160.602
C05080=1013.012,117.106,375.996,166.157,58.296,160.600
C05081=1013.016,117.355,375.979,166.161,58.285,160.599
C05082=1013.020,117.604,375.962,166.163,58.274,160.597
C05083=1013.024,117.853,375.945,166.165,58.263,160.596
C05084=1013.029,118.103,375.926,166.168,58.252,160.594
C05085=1013.032,118.352,375.909,166.171,58.241,160.593
C05086=1013.036,118.601,375.892,166.173,58.230,160.591
C05087=1013.040,118.851,375.875,166.176,58.219,160.590
C05088=1013.044,119.100,375.858,166.178,58.208,160.588
C05089=1013.048,119.349,375.841,166.181,58.197,160.587
C05090=1013.052,119.599,375.824,166.184,58.186,160.585
C05091=1013.056,119.848,375.806,166.186,58.175,160.583
C05092=1013.060,120.098,375.789,166.189,58.163,160.582
C05093=1013.064,120.347,375.772,166.191,58.153,160.581
C05094=1013.068,120.596,375.755,166.194,58.142,160.579
C05095=1013.072,120.846,375.738,166.197,58.130,160.578
C05096=1013.076,121.095,375.721,166.199,58.120,160.576
C05097=1013.080,121.345,375.704,166.203,58.108,160.575
C05098=1013.084,121.594,375.687,166.204,58.097,160.573
C05099=1013.088,121.844,375.669,166.207,58.086,160.571
C05100=1013.093,122.123,375.650,166.211,58.073,160.570
C05101=1013.097,122.402,375.630,166.213,58.061,160.568
C05102=1013.102,122.682,375.611,166.217,58.048,160.566
C05103=1013.107,122.962,375.591,166.219,58.035,160.564
C05104=1013.110,123.211,375.574,166.222,58.024,160.563
C05105=1013.114,123.460,375.557,166.225,58.013,160.562
C05106=1013.119,123.710,375.539,166.227,58.002,160.560
C05107=1013.123,123.960,375.522,166.230,57.991,160.558
C05108=1013.126,124.209,375.505,166.232,57.980,160.557
C05109=1013.131,124.457,375.487,166.235,57.968,160.555
C05110=1013.135,124.707,375.470,166.238,57.957,160.554
C05111=1013.139,124.957,375.453,166.241,57.946,160.552
C05112=1013.143,125.206,375.436,166.243,57.934,160.550
C05113=1013.147,125.456,375.418,166.246,57.923,160.549
C05114=1013.151,125.705,375.401,166.250,57.912,160.548
C05115=1013.155,125.954,375.384,166.252,57.900,160.546
C05116=1013.159,126.203,375.366,166.255,57.889,160.544
C05117=1013.164,126.453,375.349,166.257,57.877,160.543
C05118=1013.168,126.702,375.332,166.260,57.866,160.541
C05119=1013.171,126.952,375.315,166.263,57.855,160.540
C05120=1013.176,127.201,375.297,166.266,57.843,160.538
C05121=1013.180,127.450,375.280,166.269,57.832,160.537
C05122=1013.184,127.699,375.263,166.271,57.821,160.535
C05123=1013.188,127.949,375.245,166.274,57.809,160.534
C05124=1013.193,128.198,375.227,166.276,57.798,160.532
C05125=1013.197,128.447,375.210,166.280,57.787,160.530
C05126=1013.201,128.697,375.193,166.283,57.775,160.529
C05127=1013.205,128.947,375.176,166.285,57.764,160.527
C05128=1013.209,129.195,375.158,166.288,57.752,160.526
C05129=1013.213,129.446,375.140,166.292,57.741,160.524
C05130=1013.217,129.694,375.122,166.293,57.729,160.522
C05131=1013.221,129.944,375.105,166.297,57.718,160.521
C05132=1013.225,130.194,375.087,166.299,57.706,160.519
C05133=1013.229,130.442,375.069,166.302,57.695,160.518
C05134=1013.233,130.692,375.052,166.306,57.684,160.517
C05135=1013.237,130.941,375.033,166.308,57.672,160.515
C05136=1013.241,131.191,375.016,166.311,57.661,160.513
C05137=1013.245,131.440,374.998,166.313,57.650,160.512
C05138=1013.248,131.690,374.980,166.317,57.639,160.510
C05139=1013.253,131.939,374.962,166.320,57.627,160.509
C05140=1013.257,132.188,374.944,166.322,57.616,160.507
C05141=1013.261,132.438,374.926,166.325,57.604,160.505
C05142=1013.265,132.686,374.909,166.329,57.593,160.504
C05143=1013.268,132.936,374.891,166.331,57.581,160.502
C05144=1013.273,133.185,374.873,166.334,57.570,160.501
C05145=1013.276,133.435,374.855,166.337,57.558,160.499
C05146=1013.281,133.684,374.837,166.340,57.547,160.498
C05147=1013.285,133.934,374.820,166.343,57.535,160.496
C05148=1013.289,134.183,374.801,166.345,57.524,160.495
C05149=1013.293,134.432,374.783,166.348,57.513,160.493
C05150=1013.296,134.681,374.766,166.351,57.501,160.491
C05151=1013.301,134.931,374.747,166.355,57.490,160.490
C05152=1013.305,135.180,374.730,166.358,57.478,160.489
C05153=1013.309,135.430,374.712,166.360,57.467,160.487
C05154=1013.313,135.678,374.694,166.363,57.455,160.485
C05155=1013.317,135.929,374.676,166.366,57.443,160.484
C05156=1013.321,136.177,374.658,166.369,57.433,160.482
C05157=1013.325,136.427,374.639,166.372,57.421,160.481
C05158=1013.329,136.676,374.622,166.375,57.409,160.479
C05159=1013.333,136.926,374.603,166.378,57.398,160.478
C05160=1013.337,137.175,374.586,166.381,57.386,160.476
C05161=1013.341,137.424,374.567,166.384,57.375,160.475
C05162=1013.345,137.674,374.550,166.387,57.363,160.473
C05163=1013.349,137.923,374.531,166.390,57.351,160.471
C05164=1013.354,138.202,374.510,166.393,57.338,160.470
C05165=1013.358,138.482,374.491,166.396,57.326,160.468
C05166=1013.363,138.761,374.470,166.400,57.313,160.466
C05167=1013.366,139.041,374.449,166.403,57.300,160.465
C05168=1013.371,139.291,374.431,166.406,57.288,160.463
C05169=1013.375,139.540,374.413,166.410,57.277,160.461
C05170=1013.379,139.789,374.394,166.412,57.266,160.460
C05171=1013.383,140.038,374.376,166.415,57.254,160.458
C05172=1013.387,140.288,374.358,166.418,57.242,160.457
C05173=1013.390,140.537,374.339,166.422,57.231,160.455
C05174=1013.395,140.787,374.322,166.425,57.219,160.454
C05175=1013.399,141.036,374.303,166.428,57.207,160.452
C05176=1013.402,141.285,374.285,166.431,57.197,160.451
C05177=1013.407,141.535,374.266,166.434,57.185,160.449
C05178=1013.410,141.784,374.248,166.437,57.173,160.447
C05179=1013.415,142.033,374.230,166.440,57.161,160.446
C05180=1013.419,142.282,374.211,166.444,57.150,160.445
C05181=1013.423,142.531,374.193,166.447,57.138,160.443
C05182=1013.427,142.780,374.175,166.450,57.126,160.441
C05183=1013.431,143.030,374.156,166.453,57.114,160.440
C05184=1013.435,143.279,374.137,166.455,57.103,160.438
C05185=1013.439,143.528,374.120,166.459,57.092,160.437
C05186=1013.443,143.778,374.101,166.462,57.080,160.435
C05187=1013.447,144.027,374.082,166.465,57.068,160.434
C05188=1013.451,144.276,374.064,166.468,57.056,160.432
C05189=1013.455,144.526,374.046,166.471,57.045,160.430
C05190=1013.459,144.775,374.027,166.475,57.034,160.429
C05191=1013.464,145.024,374.009,166.478,57.022,160.427
C05192=1013.467,145.273,373.991,166.481,57.010,160.426
C05193=1013.471,145.523,373.972,166.484,56.998,160.424
C05194=1013.475,145.772,373.953,166.487,56.986,160.423
C05195=1013.479,146.021,373.935,166.491,56.975,160.421
C05196=1013.483,146.271,373.917,166.494,56.963,160.420
C05197=1013.487,146.520,373.898,166.497,56.952,160.418
C05198=1013.491,146.769,373.879,166.500,56.940,160.417
C05199=1013.495,147.018,373.860,166.504,56.928,160.415
C05200=1013.499,147.268,373.841,166.507,56.916,160.413
C05201=1013.503,147.517,373.823,166.509,56.906,160.412
C05202=1013.507,147.767,373.804,166.513,56.894,160.410
C05203=1013.511,148.016,373.785,166.516,56.882,160.409
C05204=1013.515,148.265,373.766,166.519,56.870,160.407
C05205=1013.519,148.514,373.748,166.522,56.858,160.406
C05206=1013.523,148.764,373.729,166.525,56.847,160.404
C05207=1013.527,149.013,373.711,166.529,56.835,160.403
C05208=1013.531,149.262,373.692,166.532,56.824,160.401
C05209=1013.535,149.511,373.673,166.535,56.812,160.400
C05210=1013.539,149.760,373.654,166.539,56.800,160.398
C05211=1013.543,150.010,373.635,166.542,56.788,160.396
C05212=1013.547,150.259,373.616,166.545,56.777,160.395
C05213=1013.551,150.509,373.597,166.548,56.765,160.393
C05214=1013.555,150.758,373.579,166.551,56.753,160.392
C05215=1013.559,151.007,373.559,166.556,56.741,160.390
C05216=1013.563,151.256,373.541,166.559,56.730,160.389
C05217=1013.566,151.505,373.522,166.563,56.718,160.388
C05218=1013.570,151.755,373.504,166.566,56.706,160.386
C05219=1013.575,152.004,373.484,166.569,56.695,160.384
C05220=1013.579,152.254,373.465,166.572,56.683,160.383
C05221=1013.583,152.502,373.446,166.576,56.671,160.381
C05222=1013.587,152.752,373.427,166.579,56.659,160.380
C05223=1013.591,153.001,373.409,166.582,56.648,160.378
C05224=1013.595,153.250,373.389,166.585,56.636,160.377
C05225=1013.599,153.500,373.370,166.589,56.624,160.375
C05226=1013.603,153.748,373.351,166.592,56.612,160.373
C05227=1013.607,153.998,373.333,166.595,56.601,160.372
C05228=1013.611,154.278,373.311,166.600,56.587,160.370
C05229=1013.615,154.557,373.289,166.604,56.574,160.369
C05230=1013.621,154.837,373.268,166.607,56.562,160.367
C05231=1013.625,155.116,373.247,166.610,56.548,160.365
C05232=1013.629,155.365,373.227,166.614,56.536,160.363
C05233=1013.633,155.615,373.209,166.618,56.524,160.362
C05234=1013.637,155.864,373.189,166.621,56.512,160.361
C05235=1013.641,156.114,373.170,166.625,56.501,160.359
C05236=1013.646,156.363,373.151,166.628,56.489,160.357
C05237=1013.648,156.612,373.132,166.631,56.477,160.356
C05238=1013.653,156.861,373.113,166.635,56.465,160.354
C05239=1013.657,157.111,373.094,166.639,56.453,160.353
C05240=1013.661,157.360,373.074,166.642,56.442,160.351
C05241=1013.665,157.609,373.056,166.645,56.430,160.350
C05242=1013.669,157.859,373.036,166.649,56.418,160.348
C05243=1013.673,158.107,373.017,166.652,56.407,160.347
C05244=1013.677,158.357,372.998,166.655,56.395,160.345
C05245=1013.681,158.606,372.978,166.659,56.383,160.344
C05246=1013.684,158.855,372.958,166.664,56.372,160.343
C05247=1013.689,159.104,372.939,166.667,56.360,160.341
C05248=1013.692,159.354,372.919,166.670,56.348,160.339
C05249=1013.696,159.604,372.899,166.674,56.337,160.338
C05250=1013.700,159.853,372.880,166.677,56.325,160.336
C05251=1013.704,160.102,372.860,166.680,56.313,160.335
C05252=1013.708,160.351,372.840,166.684,56.302,160.333
C05253=1013.711,160.600,372.820,166.687,56.290,160.332
C05254=1013.715,160.849,372.800,166.691,56.279,160.330
C05255=1013.719,161.098,372.781,166.694,56.267,160.329
C05256=1013.723,161.347,372.761,166.699,56.255,160.328
C05257=1013.727,161.596,372.741,166.702,56.244,160.326
C05258=1013.731,161.846,372.721,166.705,56.232,160.324
C05259=1013.735,162.095,372.702,166.709,56.220,160.323
C05260=1013.739,162.344,372.682,166.712,56.209,160.321
C05261=1013.742,162.594,372.662,166.715,56.197,160.320
C05262=1013.747,162.843,372.642,166.719,56.185,160.318
C05263=1013.750,163.092,372.622,166.723,56.173,160.317
C05264=1013.754,163.340,372.603,166.727,56.161,160.315
C05265=1013.757,163.590,372.583,166.730,56.150,160.314
C05266=1013.762,163.839,372.564,166.733,56.138,160.312
C05267=1013.765,164.088,372.543,166.737,56.127,160.311
C05268=1013.769,164.337,372.523,166.741,56.114,160.309
C05269=1013.773,164.586,372.504,166.745,56.103,160.308
C05270=1013.777,164.836,372.484,166.748,56.091,160.306
C05271=1013.781,165.085,372.464,166.751,56.080,160.305
C05272=1013.785,165.334,372.444,166.756,56.067,160.303
C05273=1013.789,165.583,372.425,166.759,56.056,160.302
C05274=1013.793,165.833,372.405,166.763,56.044,160.300
C05275=1013.797,166.082,372.385,166.766,56.033,160.299
C05276=1013.801,166.331,372.365,166.770,56.021,160.297
C05277=1013.804,166.580,372.345,166.774,56.009,160.296
C05278=1013.809,166.829,372.326,166.777,55.997,160.294
C05279=1013.812,167.079,372.306,166.782,55.985,160.293
C05280=1013.816,167.328,372.286,166.785,55.974,160.291
C05281=1013.821,167.577,372.265,166.789,55.962,160.290
C05282=1013.824,167.826,372.245,166.793,55.950,160.289
C05283=1013.829,168.075,372.226,166.797,55.938,160.287
C05284=1013.832,168.324,372.206,166.800,55.927,160.286
C05285=1013.837,168.574,372.186,166.804,55.915,160.284
C05286=1013.841,168.823,372.166,166.808,55.903,160.283
C05287=1013.844,169.073,372.146,166.811,55.892,160.281
C05288=1013.849,169.321,372.126,166.816,55.880,160.280
C05289=1013.853,169.570,372.106,166.819,55.867,160.278
C05290=1013.857,169.820,372.086,166.822,55.856,160.276
C05291=1013.861,170.069,372.066,166.827,55.844,160.275
C05292=1013.865,170.348,372.044,166.831,55.831,160.273
C05293=1013.870,170.628,372.021,166.835,55.817,160.272
C05294=1013.874,170.907,371.998,166.839,55.804,160.270
C05295=1013.879,171.186,371.976,166.844,55.791,160.268
C05296=1013.883,171.435,371.956,166.847,55.779,160.267
C05297=1013.887,171.685,371.936,166.852,55.767,160.265
C05298=1013.891,171.935,371.916,166.855,55.755,160.264
C05299=1013.896,172.183,371.896,166.860,55.743,160.263
C05300=1013.899,172.432,371.876,166.863,55.731,160.261
C05301=1013.904,172.681,371.856,166.867,55.719,160.259
C05302=1013.907,172.930,371.835,166.871,55.708,160.258
C05303=1013.912,173.180,371.815,166.875,55.696,160.257
C05304=1013.916,173.429,371.796,166.879,55.684,160.255
C05305=1013.920,173.679,371.775,166.883,55.672,160.254
C05306=1013.924,173.927,371.755,166.886,55.660,160.252
C05307=1013.928,174.176,371.735,166.891,55.648,160.251
C05308=1013.932,174.425,371.716,166.894,55.636,160.249
C05309=1013.937,174.675,371.695,166.899,55.624,160.248
C05310=1013.940,174.924,371.675,166.903,55.613,160.246
C05311=1013.945,175.173,371.654,166.907,55.600,160.245
C05312=1013.949,175.422,371.634,166.910,55.589,160.243
C05313=1013.954,175.672,371.614,166.915,55.577,160.242
C05314=1013.957,175.920,371.594,166.918,55.565,160.240
C05315=1013.961,176.170,371.574,166.922,55.552,160.239
C05316=1013.966,176.418,371.553,166.926,55.541,160.237
C05317=1013.969,176.668,371.533,166.931,55.529,160.236
C05318=1013.974,176.917,371.513,166.935,55.517,160.234
C05319=1013.978,177.166,371.493,166.938,55.505,160.233
C05320=1013.982,177.415,371.473,166.943,55.493,160.231
C05321=1013.987,177.664,371.452,166.946,55.481,160.230
C05322=1013.991,177.914,371.432,166.951,55.469,160.228
C05323=1013.995,178.162,371.412,166.955,55.457,160.227
C05324=1013.999,178.412,371.392,166.959,55.445,160.225
C05325=1014.003,178.661,371.371,166.963,55.433,160.224
C05326=1014.008,178.910,371.351,166.966,55.421,160.222
C05327=1014.012,179.159,371.330,166.971,55.409,160.221
C05328=1014.017,179.409,371.311,166.976,55.397,160.219
C05329=1014.021,179.657,371.290,166.979,55.385,160.218
C05330=1014.024,179.907,371.270,166.983,55.373,160.216
C05331=1014.029,180.156,371.249,166.988,55.361,160.215
C05332=1014.033,180.405,371.229,166.991,55.350,160.214
C05333=1014.038,180.654,371.209,166.996,55.337,160.212
C05334=1014.042,180.904,371.188,167.000,55.325,160.211
C05335=1014.046,181.152,371.168,167.004,55.314,160.209
C05336=1014.050,181.401,371.148,167.008,55.301,160.207
C05337=1014.055,181.651,371.127,167.013,55.289,160.206
C05338=1014.058,181.900,371.106,167.016,55.278,160.205
C05339=1014.062,182.149,371.085,167.021,55.266,160.203
C05340=1014.066,182.398,371.064,167.025,55.254,160.202
C05341=1014.071,182.647,371.043,167.029,55.243,160.200
C05342=1014.074,182.896,371.021,167.033,55.231,160.199
C05343=1014.078,183.145,371.000,167.038,55.219,160.198
C05344=1014.082,183.395,370.979,167.041,55.208,160.196
C05345=1014.086,183.644,370.958,167.046,55.196,160.195
C05346=1014.090,183.892,370.937,167.050,55.184,160.193
C05347=1014.094,184.142,370.916,167.054,55.173,160.192
C05348=1014.098,184.391,370.895,167.058,55.161,160.190
C05349=1014.102,184.640,370.873,167.063,55.149,160.189
C05350=1014.106,184.889,370.853,167.067,55.137,160.188
C05351=1014.110,185.138,370.832,167.070,55.125,160.186
C05352=1014.114,185.387,370.811,167.075,55.113,160.185
C05353=1014.117,185.636,370.789,167.079,55.102,160.183
C05354=1014.122,185.886,370.768,167.084,55.090,160.182
C05355=1014.126,186.134,370.747,167.087,55.079,160.180
C05356=1014.130,186.414,370.724,167.092,55.066,160.179
C05357=1014.134,186.693,370.700,167.097,55.052,160.177
C05358=1014.140,186.972,370.676,167.102,55.039,160.176
C05359=1014.144,187.252,370.652,167.107,55.025,160.174
C05360=1014.148,187.500,370.631,167.111,55.014,160.173
C05361=1014.152,187.750,370.609,167.116,55.002,160.171
C05362=1014.156,187.999,370.589,167.120,54.990,160.170
C05363=1014.160,188.248,370.567,167.124,54.979,160.168
C05364=1014.164,188.496,370.546,167.129,54.967,160.167
C05365=1014.168,188.746,370.524,167.134,54.955,160.166
C05366=1014.172,188.995,370.503,167.137,54.943,160.164
C05367=1014.177,189.244,370.482,167.142,54.931,160.163
C05368=1014.180,189.493,370.462,167.146,54.920,160.161
C05369=1014.184,189.743,370.440,167.150,54.908,160.160
C05370=1014.188,189.991,370.418,167.155,54.896,160.159
C05371=1014.193,190.240,370.397,167.160,54.885,160.157
C05372=1014.197,190.490,370.376,167.164,54.873,160.156
C05373=1014.201,190.739,370.355,167.168,54.861,160.154
C05374=1014.205,190.988,370.333,167.172,54.849,160.153
C05375=1014.209,191.236,370.312,167.177,54.837,160.151
C05376=1014.213,191.486,370.290,167.181,54.826,160.150
C05377=1014.217,191.734,370.269,167.186,54.814,160.149
C05378=1014.222,191.984,370.248,167.190,54.802,160.147
C05379=1014.226,192.233,370.226,167.195,54.790,160.146
C05380=1014.230,192.482,370.205,167.199,54.778,160.144
C05381=1014.234,192.731,370.183,167.203,54.767,160.143
C05382=1014.238,192.980,370.162,167.208,54.755,160.142
C05383=1014.243,193.228,370.141,167.213,54.743,160.140
C05384=1014.247,193.478,370.119,167.218,54.731,160.139
C05385=1014.251,193.727,370.098,167.222,54.719,160.137
C05386=1014.256,193.976,370.076,167.226,54.707,160.136
C05387=1014.259,194.225,370.054,167.231,54.696,160.135
C05388=1014.263,194.474,370.034,167.235,54.684,160.133
C05389=1014.268,194.723,370.012,167.240,54.672,160.132
C05390=1014.273,194.972,369.991,167.245,54.660,160.131
C05391=1014.276,195.221,369.969,167.249,54.648,160.129
C05392=1014.281,195.470,369.947,167.253,54.637,160.127
C05393=1014.286,195.719,369.926,167.258,54.625,160.126
C05394=1014.289,195.969,369.904,167.263,54.613,160.125
C05395=1014.293,196.218,369.883,167.267,54.601,160.123
C05396=1014.298,196.466,369.861,167.272,54.589,160.122
C05397=1014.303,196.716,369.840,167.277,54.577,160.121
C05398=1014.306,196.964,369.818,167.282,54.565,160.119
C05399=1014.311,197.214,369.797,167.287,54.554,160.118
C05400=1014.315,197.462,369.775,167.290,54.542,160.116
C05401=1014.320,197.712,369.754,167.295,54.530,160.115
C05402=1014.323,197.960,369.732,167.300,54.518,160.114
C05403=1014.328,198.209,369.710,167.304,54.507,160.112
C05404=1014.333,198.459,369.689,167.309,54.495,160.111
C05405=1014.337,198.708,369.666,167.314,54.482,160.109
C05406=1014.341,198.957,369.645,167.319,54.471,160.108
C05407=1014.345,199.206,369.623,167.323,54.459,160.107
C05408=1014.350,199.454,369.601,167.328,54.447,160.105
C05409=1014.354,199.704,369.579,167.333,54.436,160.104
C05410=1014.358,199.953,369.557,167.337,54.424,160.103
C05411=1014.362,200.202,369.535,167.342,54.413,160.101
C05412=1014.366,200.451,369.513,167.347,54.401,160.100
C05413=1014.370,200.700,369.490,167.352,54.389,160.099
C05414=1014.375,200.948,369.469,167.357,54.378,160.097
C05415=1014.379,201.198,369.446,167.362,54.366,160.096
C05416=1014.383,201.447,369.424,167.366,54.354,160.095
C05417=1014.387,201.696,369.403,167.371,54.342,160.093
C05418=1014.391,201.945,369.380,167.375,54.331,160.092
C05419=1014.395,202.194,369.358,167.380,54.319,160.090
C05420=1014.415,203.311,369.259,167.905,54.401,160.226
C05421=1014.420,203.543,369.236,167.909,54.392,160.225
C05422=1014.424,203.777,369.214,167.913,54.381,160.223
C05423=1014.429,204.010,369.192,167.918,54.371,160.222
C05424=1014.435,204.242,369.169,167.921,54.361,160.221
C05425=1014.439,204.475,369.147,167.926,54.351,160.220
C05426=1014.444,204.708,369.125,167.930,54.341,160.218
C05427=1014.449,204.940,369.103,167.934,54.331,160.217
C05428=1014.454,205.173,369.081,167.939,54.322,160.216
C05429=1014.460,205.422,369.056,167.943,54.311,160.215
C05430=1014.465,205.671,369.033,167.947,54.301,160.213
C05431=1014.470,205.920,369.009,167.952,54.290,160.212
C05432=1014.475,206.168,368.984,167.956,54.280,160.211
C05433=1014.481,206.418,368.960,167.960,54.269,160.210
C05434=1014.486,206.667,368.936,167.964,54.258,160.208
C05435=1014.491,206.915,368.912,167.969,54.248,160.207
C05436=1014.497,207.164,368.888,167.974,54.237,160.206
C05437=1014.502,207.413,368.863,167.978,54.227,160.204
C05438=1014.507,207.662,368.840,167.983,54.217,160.203
C05439=1014.512,207.910,368.816,167.987,54.206,160.202
C05440=1014.518,208.159,368.791,167.992,54.196,160.201
C05441=1014.523,208.408,368.767,167.996,54.185,160.199
C05442=1014.528,208.656,368.743,168.000,54.175,160.198
C05443=1014.533,208.905,368.719,168.005,54.165,160.197
C05444=1014.538,209.154,368.695,168.009,54.154,160.196
C05445=1014.544,209.403,368.671,168.014,54.144,160.194
C05446=1014.550,209.652,368.646,168.019,54.134,160.193
C05447=1014.554,209.901,368.621,168.023,54.124,160.192
C05448=1014.559,210.149,368.597,168.027,54.113,160.191
C05449=1014.565,210.398,368.573,168.032,54.103,160.190
C05450=1014.570,210.646,368.548,168.036,54.093,160.188
C05451=1014.575,210.895,368.524,168.040,54.083,160.187
